# B&R Automation Studio project MotionTestBenchMaster (part 29)

```iecst
								VAR_RNS_SEQ.Device.PPB209_PID.PID_Enable := FALSE;                                      (* STEP: 0 PPB209*)
								VAR_RNS_SEQ.Device.PPB209_PID.PID_Mode := FALSE;
								VAR_RNS_SEQ.Device.PPB209_PID.Auto_SP_Value := 0;
								VAR_RNS_SEQ.Device.PPB209_PID.FIX_Value := 0;

								VAR_RNS_SEQ.Device.RVB202_PID.PID_Enable := FALSE;                                      (* STEP: 0 *)
								VAR_RNS_SEQ.Device.RVB202_PID.PID_Mode := FALSE;
								VAR_RNS_SEQ.Device.RVB202_PID.Auto_SP_Value := 0;
								VAR_RNS_SEQ.Device.RVB202_PID.FIX_Value := 0;

								VAR_RNS_SEQ.Device.FSB220.ALR := FALSE;                                                 (* STEP: 0 FSB220*)
								VAR_RNS_SEQ.Device.FSB220.WAIT_OFF := FALSE;
								VAR_RNS_SEQ.Device.FSB220.WAIT_ON := FALSE;

								VAR_RNS_SEQ.Device.LSB209.ALR := FALSE;                                                 (* STEP: 0 LSB209*)
								VAR_RNS_SEQ.Device.LSB209.WAIT_OFF := FALSE;
								VAR_RNS_SEQ.Device.LSB209.WAIT_ON := FALSE;

								VAR_RNS_SEQ.Device.LSB210.ALR := FALSE;                                                 (* STEP: 0 LSB210*)
								VAR_RNS_SEQ.Device.LSB210.WAIT_OFF := FALSE;
								VAR_RNS_SEQ.Device.LSB210.WAIT_ON := FALSE;

								VAR_RNS_SEQ.Device.LSB299.ALR := FALSE;                                                 (* STEP: 0 *)
								VAR_RNS_SEQ.Device.LSB299.WAIT_OFF := FALSE;
								VAR_RNS_SEQ.Device.LSB299.WAIT_ON := FALSE;

								VAR_RNS_SEQ.Device.FSB201.ALR := FALSE;                                                 (* STEP: 0 FSB201*)
								VAR_RNS_SEQ.Device.FSB201.WAIT_OFF := FALSE;
								VAR_RNS_SEQ.Device.FSB201.WAIT_ON := FALSE;

								VAR_RNS_SEQ.Device.FTB201.ALR_HighLimitEn := FALSE;                                     (* STEP: 0 FTB201*)
								VAR_RNS_SEQ.Device.FTB201.ALR_HighLimitSP := 0;
								VAR_RNS_SEQ.Device.FTB201.ALR_LowLimitEn := FALSE;
								VAR_RNS_SEQ.Device.FTB201.ALR_LowLimitSP := 0;
								VAR_RNS_SEQ.Device.FTB201.SP := 0;
								VAR_RNS_SEQ.Device.FTB201.CMP := 0;
								VAR_RNS_SEQ.Device.FTB201.MinDev := 0;
								VAR_RNS_SEQ.Device.FTB201.MaxDev := 0;

								VAR_RNS_SEQ.Device.FTB202.ALR_HighLimitEn := FALSE;                                     (* STEP: 0 FTB202*)
								VAR_RNS_SEQ.Device.FTB202.ALR_HighLimitSP := 0;
								VAR_RNS_SEQ.Device.FTB202.ALR_LowLimitEn := FALSE;
								VAR_RNS_SEQ.Device.FTB202.ALR_LowLimitSP := 0;
								VAR_RNS_SEQ.Device.FTB202.SP := 0;
								VAR_RNS_SEQ.Device.FTB202.CMP := 0;
								VAR_RNS_SEQ.Device.FTB202.MinDev := 0;
								VAR_RNS_SEQ.Device.FTB202.MaxDev := 0;

								VAR_RNS_SEQ.Device.PTB220.ALR_HighLimitEn := FALSE;                                     (* STEP: 0 PTB220*)
								VAR_RNS_SEQ.Device.PTB220.ALR_HighLimitSP := 0;
								VAR_RNS_SEQ.Device.PTB220.ALR_LowLimitEn := FALSE;
								VAR_RNS_SEQ.Device.PTB220.ALR_LowLimitSP := 0;
								VAR_RNS_SEQ.Device.PTB220.SP := 0;
								VAR_RNS_SEQ.Device.PTB220.CMP := 0;
								VAR_RNS_SEQ.Device.PTB220.MinDev := 0;
								VAR_RNS_SEQ.Device.PTB220.MaxDev := 0;

								VAR_RNS_SEQ.Device.PTB270.ALR_HighLimitEn := FALSE;                                     (* STEP: 0 PTB270*)
								VAR_RNS_SEQ.Device.PTB270.ALR_HighLimitSP := 0;
								VAR_RNS_SEQ.Device.PTB270.ALR_LowLimitEn := FALSE;
								VAR_RNS_SEQ.Device.PTB270.ALR_LowLimitSP := 0;
								VAR_RNS_SEQ.Device.PTB270.SP := 0;
								VAR_RNS_SEQ.Device.PTB270.CMP := 0;
								VAR_RNS_SEQ.Device.PTB270.MinDev := 0;
								VAR_RNS_SEQ.Device.PTB270.MaxDev := 0;

								VAR_RNS_SEQ.Device.LTB202.ALR_HighLimitEn := FALSE;                                     (* STEP: 0 LTB202*)
								VAR_RNS_SEQ.Device.LTB202.ALR_HighLimitSP := 0;
								VAR_RNS_SEQ.Device.LTB202.ALR_LowLimitEn := FALSE;
								VAR_RNS_SEQ.Device.LTB202.ALR_LowLimitSP := 0;
								VAR_RNS_SEQ.Device.LTB202.SP := 0;
								VAR_RNS_SEQ.Device.LTB202.CMP := 0;
								VAR_RNS_SEQ.Device.LTB202.MinDev := 0;
								VAR_RNS_SEQ.Device.LTB202.MaxDev := 0;

								VAR_RNS_SEQ.Device.PTB290.ALR_HighLimitEn := FALSE;                                     (* STEP: 0 PTB290*)
								VAR_RNS_SEQ.Device.PTB290.ALR_HighLimitSP := 0;
								VAR_RNS_SEQ.Device.PTB290.ALR_LowLimitEn := FALSE;
								VAR_RNS_SEQ.Device.PTB290.ALR_LowLimitSP := 0;
								VAR_RNS_SEQ.Device.PTB290.SP := 0;
								VAR_RNS_SEQ.Device.PTB290.CMP := 0;
								VAR_RNS_SEQ.Device.PTB290.MinDev := 0;
								VAR_RNS_SEQ.Device.PTB290.MaxDev := 0;

								VAR_RNS_SEQ.Mem.ContainersStop := TRUE;                                                (* STEP: 0 *)
								VAR_RNS_SEQ.Mem.ControlInsercion := FALSE;                                              (* STEP: 0 *)
								VAR_RNS_SEQ.Mem.ControlContinous := FALSE;                                              (* STEP: 0 *)
								VAR_RNS_SEQ.Mem.PBAbortEnable := FALSE;                                                 (* STEP: 0 PB Abort Sequence Enable*)
								VAR_RNS_SEQ.Mem.PBStopEnable := TRUE;                                                  (* STEP: 0 PB Stop Sequence Enable*)
								VAR_RNS_SEQ.Mem.PBStartEnable := FALSE;                                                  (* STEP: 0 PB Start Sequence Enable*)
								VAR_RNS_SEQ.Mem.ByPassed := FALSE;                                                      (* STEP: 0 *)
								VAR_RNS_SEQ.Mem.InsercionDevice := FALSE;                                               (* STEP: 0 *)
								VAR_RNS_SEQ.Mem.AirTreatmentControl := FALSE;                                           (* STEP: 0 *)
								VAR_RNS_SEQ.Mem.WaterTreatmentControl := FALSE;                                         (* STEP: 0 *)
								VAR_RNS_SEQ.Mem.SpeedReductionControl := FALSE;                                         (* STEP: 0 *)
								VAR_RNS_SEQ.Mem.ByPassRequest := FALSE;                                                 (* STEP: 0 *)
								VAR_RNS_SEQ.Mem.CopAfterCipRequest := FALSE;                                            (* STEP: 0 *)
								VAR_RNS_SEQ.Mem.NoBoNoSprayInsercion := FALSE;                                          (* STEP: 0 *)

								VAR_RNS_SEQ.ITC.WTT_ProductRequest := FALSE;                                            (* STEP: 0 *)
								VAR_RNS_SEQ.ITC.WTT_ProductionRunning := FALSE;

							36: (*MOTORIZATION - Waiting for Machine Stop - Disabling Axis*) //RnsDisable

								VAR_RNS_SEQ.Device.AVB224.AutoCnd := TRUE;                                              (* STEP: 0 AVB224*)
								VAR_RNS_SEQ.Device.AVB224.EnableCnd := FALSE;
								VAR_RNS_SEQ.Device.AVB228.AutoCnd := FALSE;                                             (* STEP: 0 AVB228*)
								VAR_RNS_SEQ.Device.AVB228.EnableCnd := FALSE;
								VAR_RNS_SEQ.Device.AVB234.AutoCnd := TRUE;                                              (* STEP: 0 AVB234*)
								VAR_RNS_SEQ.Device.AVB234.EnableCnd := FALSE;
								VAR_RNS_SEQ.Device.AVB261.AutoCnd := FALSE;                                             (* STEP: 0 AVB261*)
								VAR_RNS_SEQ.Device.AVB261.EnableCnd := FALSE;
								VAR_RNS_SEQ.Device.AVB264.AutoCnd := FALSE;                                             (* STEP: 0 AVB264*)
								VAR_RNS_SEQ.Device.AVB264.EnableCnd := FALSE;
								VAR_RNS_SEQ.Device.AVB265.AutoCnd := FALSE;                                             (* STEP: 0 AVB265*)
								VAR_RNS_SEQ.Device.AVB265.EnableCnd := FALSE;
								VAR_RNS_SEQ.Device.AVB266.AutoCnd := FALSE;                                             (* STEP: 0 AVB266*)
								VAR_RNS_SEQ.Device.AVB266.EnableCnd := FALSE;
								VAR_RNS_SEQ.Device.AVB267.AutoCnd := TRUE;                                              (* STEP: 0 AVB267*)
								VAR_RNS_SEQ.Device.AVB267.EnableCnd := FALSE;
								VAR_RNS_SEQ.Device.AVB268.AutoCnd := TRUE;                                              (* STEP: 0 AVB268*)
								VAR_RNS_SEQ.Device.AVB268.EnableCnd := FALSE;
								VAR_RNS_SEQ.Device.AVB273.AutoCnd := FALSE;                                             (* STEP: 0 AVB273*)
								VAR_RNS_SEQ.Device.AVB273.EnableCnd := FALSE;
								VAR_RNS_SEQ.Device.AVB294.AutoCnd := FALSE;                                             (* STEP: 0 AVB294*)
								VAR_RNS_SEQ.Device.AVB294.EnableCnd := FALSE;

								VAR_RNS_SEQ.Device.PPB209_PID.PID_Enable := FALSE;                                      (* STEP: 0 PPB209*)
								VAR_RNS_SEQ.Device.PPB209_PID.PID_Mode := FALSE;
								VAR_RNS_SEQ.Device.PPB209_PID.Auto_SP_Value := 0;
								VAR_RNS_SEQ.Device.PPB209_PID.FIX_Value := 0;

								VAR_RNS_SEQ.Device.RVB202_PID.PID_Enable := FALSE;                                      (* STEP: 0 *)
								VAR_RNS_SEQ.Device.RVB202_PID.PID_Mode := FALSE;
								VAR_RNS_SEQ.Device.RVB202_PID.Auto_SP_Value := 0;
								VAR_RNS_SEQ.Device.RVB202_PID.FIX_Value := 0;

								VAR_RNS_SEQ.Device.FSB220.ALR := FALSE;                                                 (* STEP: 0 FSB220*)
								VAR_RNS_SEQ.Device.FSB220.WAIT_OFF := FALSE;
								VAR_RNS_SEQ.Device.FSB220.WAIT_ON := FALSE;

								VAR_RNS_SEQ.Device.LSB209.ALR := FALSE;                                                 (* STEP: 0 LSB209*)
								VAR_RNS_SEQ.Device.LSB209.WAIT_OFF := FALSE;
								VAR_RNS_SEQ.Device.LSB209.WAIT_ON := FALSE;

								VAR_RNS_SEQ.Device.LSB210.ALR := FALSE;                                                 (* STEP: 0 LSB210*)
								VAR_RNS_SEQ.Device.LSB210.WAIT_OFF := FALSE;
								VAR_RNS_SEQ.Device.LSB210.WAIT_ON := FALSE;

								VAR_RNS_SEQ.Device.LSB299.ALR := FALSE;                                                 (* STEP: 0 *)
								VAR_RNS_SEQ.Device.LSB299.WAIT_OFF := FALSE;
								VAR_RNS_SEQ.Device.LSB299.WAIT_ON := FALSE;

								VAR_RNS_SEQ.Device.FSB201.ALR := FALSE;                                                 (* STEP: 0 FSB201*)
								VAR_RNS_SEQ.Device.FSB201.WAIT_OFF := FALSE;
								VAR_RNS_SEQ.Device.FSB201.WAIT_ON := FALSE;

								VAR_RNS_SEQ.Device.FTB201.ALR_HighLimitEn := FALSE;                                     (* STEP: 0 FTB201*)
								VAR_RNS_SEQ.Device.FTB201.ALR_HighLimitSP := 0;
								VAR_RNS_SEQ.Device.FTB201.ALR_LowLimitEn := FALSE;
								VAR_RNS_SEQ.Device.FTB201.ALR_LowLimitSP := 0;
								VAR_RNS_SEQ.Device.FTB201.SP := 0;
								VAR_RNS_SEQ.Device.FTB201.CMP := 0;
								VAR_RNS_SEQ.Device.FTB201.MinDev := 0;
								VAR_RNS_SEQ.Device.FTB201.MaxDev := 0;

								VAR_RNS_SEQ.Device.FTB202.ALR_HighLimitEn := FALSE;                                     (* STEP: 0 FTB202*)
								VAR_RNS_SEQ.Device.FTB202.ALR_HighLimitSP := 0;
								VAR_RNS_SEQ.Device.FTB202.ALR_LowLimitEn := FALSE;
								VAR_RNS_SEQ.Device.FTB202.ALR_LowLimitSP := 0;
								VAR_RNS_SEQ.Device.FTB202.SP := 0;
								VAR_RNS_SEQ.Device.FTB202.CMP := 0;
								VAR_RNS_SEQ.Device.FTB202.MinDev := 0;
								VAR_RNS_SEQ.Device.FTB202.MaxDev := 0;

								VAR_RNS_SEQ.Device.PTB220.ALR_HighLimitEn := FALSE;                                     (* STEP: 0 PTB220*)
								VAR_RNS_SEQ.Device.PTB220.ALR_HighLimitSP := 0;
								VAR_RNS_SEQ.Device.PTB220.ALR_LowLimitEn := FALSE;
								VAR_RNS_SEQ.Device.PTB220.ALR_LowLimitSP := 0;
								VAR_RNS_SEQ.Device.PTB220.SP := 0;
								VAR_RNS_SEQ.Device.PTB220.CMP := 0;
								VAR_RNS_SEQ.Device.PTB220.MinDev := 0;
								VAR_RNS_SEQ.Device.PTB220.MaxDev := 0;

								VAR_RNS_SEQ.Device.PTB270.ALR_HighLimitEn := FALSE;                                     (* STEP: 0 PTB270*)
								VAR_RNS_SEQ.Device.PTB270.ALR_HighLimitSP := 0;
								VAR_RNS_SEQ.Device.PTB270.ALR_LowLimitEn := FALSE;
								VAR_RNS_SEQ.Device.PTB270.ALR_LowLimitSP := 0;
								VAR_RNS_SEQ.Device.PTB270.SP := 0;
								VAR_RNS_SEQ.Device.PTB270.CMP := 0;
								VAR_RNS_SEQ.Device.PTB270.MinDev := 0;
								VAR_RNS_SEQ.Device.PTB270.MaxDev := 0;

								VAR_RNS_SEQ.Device.LTB202.ALR_HighLimitEn := FALSE;                                     (* STEP: 0 LTB202*)
								VAR_RNS_SEQ.Device.LTB202.ALR_HighLimitSP := 0;
								VAR_RNS_SEQ.Device.LTB202.ALR_LowLimitEn := FALSE;
								VAR_RNS_SEQ.Device.LTB202.ALR_LowLimitSP := 0;
								VAR_RNS_SEQ.Device.LTB202.SP := 0;
								VAR_RNS_SEQ.Device.LTB202.CMP := 0;
								VAR_RNS_SEQ.Device.LTB202.MinDev := 0;
								VAR_RNS_SEQ.Device.LTB202.MaxDev := 0;

								VAR_RNS_SEQ.Device.PTB290.ALR_HighLimitEn := FALSE;                                     (* STEP: 0 PTB290*)
								VAR_RNS_SEQ.Device.PTB290.ALR_HighLimitSP := 0;
								VAR_RNS_SEQ.Device.PTB290.ALR_LowLimitEn := FALSE;
								VAR_RNS_SEQ.Device.PTB290.ALR_LowLimitSP := 0;
								VAR_RNS_SEQ.Device.PTB290.SP := 0;
								VAR_RNS_SEQ.Device.PTB290.CMP := 0;
								VAR_RNS_SEQ.Device.PTB290.MinDev := 0;
								VAR_RNS_SEQ.Device.PTB290.MaxDev := 0;

								VAR_RNS_SEQ.Mem.ContainersStop := TRUE;                                                (* STEP: 0 *)
								VAR_RNS_SEQ.Mem.ControlInsercion := FALSE;                                              (* STEP: 0 *)
								VAR_RNS_SEQ.Mem.ControlContinous := FALSE;                                              (* STEP: 0 *)
								VAR_RNS_SEQ.Mem.PBAbortEnable := FALSE;                                                 (* STEP: 0 PB Abort Sequence Enable*)
								VAR_RNS_SEQ.Mem.PBStopEnable := TRUE;                                                  (* STEP: 0 PB Stop Sequence Enable*)
								VAR_RNS_SEQ.Mem.PBStartEnable := TRUE;                                                  (* STEP: 0 PB Start Sequence Enable*)
								VAR_RNS_SEQ.Mem.ByPassed := FALSE;                                                      (* STEP: 0 *)
								VAR_RNS_SEQ.Mem.InsercionDevice := FALSE;                                               (* STEP: 0 *)
								VAR_RNS_SEQ.Mem.AirTreatmentControl := FALSE;                                           (* STEP: 0 *)
								VAR_RNS_SEQ.Mem.WaterTreatmentControl := FALSE;                                         (* STEP: 0 *)
								VAR_RNS_SEQ.Mem.SpeedReductionControl := FALSE;                                         (* STEP: 0 *)
								VAR_RNS_SEQ.Mem.ByPassRequest := FALSE;                                                 (* STEP: 0 *)
								VAR_RNS_SEQ.Mem.CopAfterCipRequest := FALSE;                                            (* STEP: 0 *)
								VAR_RNS_SEQ.Mem.NoBoNoSprayInsercion := FALSE;                                          (* STEP: 0 *)

								VAR_RNS_SEQ.ITC.WTT_ProductRequest := FALSE;                                            (* STEP: 0 *)
								VAR_RNS_SEQ.ITC.WTT_ProductionRunning := FALSE;

						37..39: (* Spare Steps *)

						40: (* CIP - Wait Condition *)

                               VAR_RNS_SEQ.Device.AVB224.AutoCnd := FALSE;                                             (* STEP: 40 AVB224*)
                               VAR_RNS_SEQ.Device.AVB224.EnableCnd := FALSE;
                               VAR_RNS_SEQ.Device.AVB228.AutoCnd := FALSE;                                             (* STEP: 40 AVB228*)
                               VAR_RNS_SEQ.Device.AVB228.EnableCnd := FALSE;
                               VAR_RNS_SEQ.Device.AVB234.AutoCnd := FALSE;                                             (* STEP: 40 AVB234*)
                               VAR_RNS_SEQ.Device.AVB234.EnableCnd := FALSE;
                               VAR_RNS_SEQ.Device.AVB261.AutoCnd := TRUE;                                             (* STEP: 40 AVB261*)
                               VAR_RNS_SEQ.Device.AVB261.EnableCnd := FALSE;
                               VAR_RNS_SEQ.Device.AVB264.AutoCnd := FALSE;                                             (* STEP: 40 AVB264*)
                               VAR_RNS_SEQ.Device.AVB264.EnableCnd := FALSE;
                               VAR_RNS_SEQ.Device.AVB265.AutoCnd := FALSE;                                             (* STEP: 40 AVB265*)
                               VAR_RNS_SEQ.Device.AVB265.EnableCnd := FALSE;
                               VAR_RNS_SEQ.Device.AVB266.AutoCnd := TRUE;                                              (* STEP: 40 AVB266*)
                               VAR_RNS_SEQ.Device.AVB266.EnableCnd := FALSE;
                               VAR_RNS_SEQ.Device.AVB267.AutoCnd := FALSE;                                             (* STEP: 40 AVB267*)
                               VAR_RNS_SEQ.Device.AVB267.EnableCnd := FALSE;
                               VAR_RNS_SEQ.Device.AVB268.AutoCnd := FALSE;                                             (* STEP: 40 AVB268*)
                               VAR_RNS_SEQ.Device.AVB268.EnableCnd := FALSE;
                               VAR_RNS_SEQ.Device.AVB273.AutoCnd := FALSE;                                             (* STEP: 40 AVB273*)
                               VAR_RNS_SEQ.Device.AVB273.EnableCnd := FALSE;
                               VAR_RNS_SEQ.Device.AVB294.AutoCnd := FALSE;                                             (* STEP: 40 AVB294*)
                               VAR_RNS_SEQ.Device.AVB294.EnableCnd := FALSE;

                               VAR_RNS_SEQ.Device.PPB209_PID.PID_Enable := FALSE;                                      (* STEP: 40 PPB209*)
                               VAR_RNS_SEQ.Device.PPB209_PID.PID_Mode := FALSE;
                               VAR_RNS_SEQ.Device.PPB209_PID.Auto_SP_Value := 0;
                               VAR_RNS_SEQ.Device.PPB209_PID.FIX_Value := 0;

                               VAR_RNS_SEQ.Device.RVB202_PID.PID_Enable := TRUE;                                       (* STEP: 40 *)
                               VAR_RNS_SEQ.Device.RVB202_PID.PID_Mode := FALSE;
                               VAR_RNS_SEQ.Device.RVB202_PID.Auto_SP_Value := 0;
                               VAR_RNS_SEQ.Device.RVB202_PID.FIX_Value := HMI_PAM_1._093;

                               VAR_RNS_SEQ.Device.FSB220.ALR := FALSE;                                                 (* STEP: 40 FSB220*)
                               VAR_RNS_SEQ.Device.FSB220.WAIT_OFF := FALSE;
                               VAR_RNS_SEQ.Device.FSB220.WAIT_ON := FALSE;

                               VAR_RNS_SEQ.Device.LSB209.ALR := FALSE;                                                 (* STEP: 40 LSB209*)
                               VAR_RNS_SEQ.Device.LSB209.WAIT_OFF := FALSE;
                               VAR_RNS_SEQ.Device.LSB209.WAIT_ON := FALSE;

                               VAR_RNS_SEQ.Device.LSB210.ALR := FALSE;                                                 (* STEP: 40 LSB210*)
                               VAR_RNS_SEQ.Device.LSB210.WAIT_OFF := FALSE;
                               VAR_RNS_SEQ.Device.LSB210.WAIT_ON := FALSE;

                               VAR_RNS_SEQ.Device.LSB299.ALR := FALSE;                                                 (* STEP: 40 *)
                               VAR_RNS_SEQ.Device.LSB299.WAIT_OFF := FALSE;
                               VAR_RNS_SEQ.Device.LSB299.WAIT_ON := FALSE;

                               VAR_RNS_SEQ.Device.FSB201.ALR := FALSE;                                                 (* STEP: 40 FSB201*)
                               VAR_RNS_SEQ.Device.FSB201.WAIT_OFF := FALSE;
                               VAR_RNS_SEQ.Device.FSB201.WAIT_ON := FALSE;

                               VAR_RNS_SEQ.Device.FTB201.ALR_HighLimitEn := FALSE;                                     (* STEP: 40 FTB201*)
                               VAR_RNS_SEQ.Device.FTB201.ALR_HighLimitSP := 0;
                               VAR_RNS_SEQ.Device.FTB201.ALR_LowLimitEn := FALSE;
                               VAR_RNS_SEQ.Device.FTB201.ALR_LowLimitSP := 0;
                               VAR_RNS_SEQ.Device.FTB201.SP := 0;
                               VAR_RNS_SEQ.Device.FTB201.CMP := 0;
                               VAR_RNS_SEQ.Device.FTB201.MinDev := 0;
                               VAR_RNS_SEQ.Device.FTB201.MaxDev := 0;

                               VAR_RNS_SEQ.Device.FTB202.ALR_HighLimitEn := FALSE;                                     (* STEP: 40 FTB202*)
                               VAR_RNS_SEQ.Device.FTB202.ALR_HighLimitSP := 0;
                               VAR_RNS_SEQ.Device.FTB202.ALR_LowLimitEn := FALSE;
                               VAR_RNS_SEQ.Device.FTB202.ALR_LowLimitSP := 0;
                               VAR_RNS_SEQ.Device.FTB202.SP := 0;
                               VAR_RNS_SEQ.Device.FTB202.CMP := 0;
                               VAR_RNS_SEQ.Device.FTB202.MinDev := 0;
                               VAR_RNS_SEQ.Device.FTB202.MaxDev := 0;

                               VAR_RNS_SEQ.Device.PTB220.ALR_HighLimitEn := FALSE;                                     (* STEP: 40 PTB220*)
                               VAR_RNS_SEQ.Device.PTB220.ALR_HighLimitSP := 0;
                               VAR_RNS_SEQ.Device.PTB220.ALR_LowLimitEn := FALSE;
                               VAR_RNS_SEQ.Device.PTB220.ALR_LowLimitSP := 0;
                               VAR_RNS_SEQ.Device.PTB220.SP := 0;
                               VAR_RNS_SEQ.Device.PTB220.CMP := 0;
                               VAR_RNS_SEQ.Device.PTB220.MinDev := 0;
                               VAR_RNS_SEQ.Device.PTB220.MaxDev := 0;

                               VAR_RNS_SEQ.Device.PTB270.ALR_HighLimitEn := FALSE;                                     (* STEP: 40 PTB270*)
                               VAR_RNS_SEQ.Device.PTB270.ALR_HighLimitSP := 0;
                               VAR_RNS_SEQ.Device.PTB270.ALR_LowLimitEn := FALSE;
                               VAR_RNS_SEQ.Device.PTB270.ALR_LowLimitSP := 0;
                               VAR_RNS_SEQ.Device.PTB270.SP := 0;
                               VAR_RNS_SEQ.Device.PTB270.CMP := 0;
                               VAR_RNS_SEQ.Device.PTB270.MinDev := 0;
                               VAR_RNS_SEQ.Device.PTB270.MaxDev := 0;

                               VAR_RNS_SEQ.Device.LTB202.ALR_HighLimitEn := FALSE;                                     (* STEP: 40 LTB202*)
                               VAR_RNS_SEQ.Device.LTB202.ALR_HighLimitSP := 0;
                               VAR_RNS_SEQ.Device.LTB202.ALR_LowLimitEn := FALSE;
                               VAR_RNS_SEQ.Device.LTB202.ALR_LowLimitSP := 0;
                               VAR_RNS_SEQ.Device.LTB202.SP := 0;
                               VAR_RNS_SEQ.Device.LTB202.CMP := 0;
                               VAR_RNS_SEQ.Device.LTB202.MinDev := 0;
                               VAR_RNS_SEQ.Device.LTB202.MaxDev := 0;

                               VAR_RNS_SEQ.Device.PTB290.ALR_HighLimitEn := FALSE;                                     (* STEP: 40 PTB290*)
                               VAR_RNS_SEQ.Device.PTB290.ALR_HighLimitSP := 0;
                               VAR_RNS_SEQ.Device.PTB290.ALR_LowLimitEn := FALSE;
                               VAR_RNS_SEQ.Device.PTB290.ALR_LowLimitSP := 0;
                               VAR_RNS_SEQ.Device.PTB290.SP := 0;
                               VAR_RNS_SEQ.Device.PTB290.CMP := 0;
                               VAR_RNS_SEQ.Device.PTB290.MinDev := 0;
                               VAR_RNS_SEQ.Device.PTB290.MaxDev := 0;

                               VAR_RNS_SEQ.Mem.ContainersStop := TRUE;                                                 (* STEP: 40 *)
                               VAR_RNS_SEQ.Mem.ControlInsercion := FALSE;                                              (* STEP: 40 *)
                               VAR_RNS_SEQ.Mem.ControlContinous := FALSE;                                              (* STEP: 40 *)
                               VAR_RNS_SEQ.Mem.PBAbortEnable := FALSE;                                                 (* STEP: 40 PB Abort Sequence Enable*)
                               VAR_RNS_SEQ.Mem.PBStopEnable := TRUE;                                                   (* STEP: 40 PB Stop Sequence Enable*)
                               VAR_RNS_SEQ.Mem.PBStartEnable := FALSE;                                                 (* STEP: 40 PB Start Sequence Enable*)
                               VAR_RNS_SEQ.Mem.ByPassed := FALSE;                                                      (* STEP: 40 *)
                               VAR_RNS_SEQ.Mem.InsercionDevice := FALSE;                                               (* STEP: 40 *)
                               VAR_RNS_SEQ.Mem.AirTreatmentControl := FALSE;                                           (* STEP: 40 *)
                               VAR_RNS_SEQ.Mem.WaterTreatmentControl := FALSE;                                         (* STEP: 40 *)
                               VAR_RNS_SEQ.Mem.SpeedReductionControl := FALSE;                                         (* STEP: 40 *)
                               VAR_RNS_SEQ.Mem.ByPassRequest := FALSE;                                                 (* STEP: 40 *)
                               VAR_RNS_SEQ.Mem.CopAfterCipRequest := FALSE;                                            (* STEP: 40 *)
                               VAR_RNS_SEQ.Mem.NoBoNoSprayInsercion := FALSE;                                          (* STEP: 40 *)

                               VAR_RNS_SEQ.ITC.WTT_ProductRequest := TRUE;                                             (* STEP: 40 *)
                               VAR_RNS_SEQ.ITC.WTT_ProductionRunning := FALSE;                                         (* STEP: 40 *)

                       41: (* CIP - Execution *)

                               VAR_RNS_SEQ.Device.AVB224.AutoCnd := FALSE;                                             (* STEP: 41 AVB224*)
                               VAR_RNS_SEQ.Device.AVB224.EnableCnd := FALSE;
                               VAR_RNS_SEQ.Device.AVB228.AutoCnd := FALSE;                                             (* STEP: 41 AVB228*)
                               VAR_RNS_SEQ.Device.AVB228.EnableCnd := FALSE;
                               VAR_RNS_SEQ.Device.AVB234.AutoCnd := FALSE;                                             (* STEP: 41 AVB234*)
                               VAR_RNS_SEQ.Device.AVB234.EnableCnd := FALSE;
                               VAR_RNS_SEQ.Device.AVB261.AutoCnd := TRUE;                                              (* STEP: 41 AVB261*)
                               VAR_RNS_SEQ.Device.AVB261.EnableCnd := FALSE;
                               VAR_RNS_SEQ.Device.AVB264.AutoCnd := FALSE;                                             (* STEP: 41 AVB264*)
                               VAR_RNS_SEQ.Device.AVB264.EnableCnd := FALSE;
                               VAR_RNS_SEQ.Device.AVB265.AutoCnd := TRUE;                                              (* STEP: 41 AVB265*)
                               VAR_RNS_SEQ.Device.AVB265.EnableCnd := FALSE;
                               VAR_RNS_SEQ.Device.AVB266.AutoCnd := TRUE;                                              (* STEP: 41 AVB266*)
                               VAR_RNS_SEQ.Device.AVB266.EnableCnd := FALSE;
                               VAR_RNS_SEQ.Device.AVB267.AutoCnd := TRUE;                                              (* STEP: 41 AVB267*)
                               VAR_RNS_SEQ.Device.AVB267.EnableCnd := FALSE;
                               VAR_RNS_SEQ.Device.AVB268.AutoCnd := TRUE;                                              (* STEP: 41 AVB268*)
                               VAR_RNS_SEQ.Device.AVB268.EnableCnd := TRUE;
                               VAR_RNS_SEQ.Device.AVB273.AutoCnd := FALSE;                                             (* STEP: 41 AVB273*)
                               VAR_RNS_SEQ.Device.AVB273.EnableCnd := FALSE;
                               VAR_RNS_SEQ.Device.AVB294.AutoCnd := TRUE;                                              (* STEP: 41 AVB294*)
                               VAR_RNS_SEQ.Device.AVB294.EnableCnd := TRUE;

                               VAR_RNS_SEQ.Device.PPB209_PID.PID_Enable := FALSE;                                      (* STEP: 41 PPB209*)
                               VAR_RNS_SEQ.Device.PPB209_PID.PID_Mode := FALSE;
                               VAR_RNS_SEQ.Device.PPB209_PID.Auto_SP_Value := 0;
                               VAR_RNS_SEQ.Device.PPB209_PID.FIX_Value := 0;

                               VAR_RNS_SEQ.Device.RVB202_PID.PID_Enable := TRUE;                                       (* STEP: 41 *)
                               VAR_RNS_SEQ.Device.RVB202_PID.PID_Mode := FALSE;
                               VAR_RNS_SEQ.Device.RVB202_PID.Auto_SP_Value := 0;
                               VAR_RNS_SEQ.Device.RVB202_PID.FIX_Value := HMI_PAM_1._093;

                               VAR_RNS_SEQ.Device.FSB220.ALR := FALSE;                                                 (* STEP: 41 FSB220*)
                               VAR_RNS_SEQ.Device.FSB220.WAIT_OFF := FALSE;
                               VAR_RNS_SEQ.Device.FSB220.WAIT_ON := FALSE;

                               VAR_RNS_SEQ.Device.LSB209.ALR := FALSE;                                                 (* STEP: 41 LSB209*)
                               VAR_RNS_SEQ.Device.LSB209.WAIT_OFF := FALSE;
                               VAR_RNS_SEQ.Device.LSB209.WAIT_ON := FALSE;

                               VAR_RNS_SEQ.Device.LSB210.ALR := FALSE;                                                 (* STEP: 41 LSB210*)
                               VAR_RNS_SEQ.Device.LSB210.WAIT_OFF := FALSE;
                               VAR_RNS_SEQ.Device.LSB210.WAIT_ON := FALSE;

                               VAR_RNS_SEQ.Device.LSB299.ALR := FALSE;                                                 (* STEP: 41 *)
                               VAR_RNS_SEQ.Device.LSB299.WAIT_OFF := FALSE;
                               VAR_RNS_SEQ.Device.LSB299.WAIT_ON := FALSE;

                               VAR_RNS_SEQ.Device.FSB201.ALR := FALSE;                                                 (* STEP: 41 FSB201*)
                               VAR_RNS_SEQ.Device.FSB201.WAIT_OFF := FALSE;
                               VAR_RNS_SEQ.Device.FSB201.WAIT_ON := FALSE;

                               VAR_RNS_SEQ.Device.FTB201.ALR_HighLimitEn := FALSE;                                     (* STEP: 41 FTB201*)
                               VAR_RNS_SEQ.Device.FTB201.ALR_HighLimitSP := 0;
                               VAR_RNS_SEQ.Device.FTB201.ALR_LowLimitEn := FALSE;
                               VAR_RNS_SEQ.Device.FTB201.ALR_LowLimitSP := 0;
                               VAR_RNS_SEQ.Device.FTB201.SP := 0;
                               VAR_RNS_SEQ.Device.FTB201.CMP := 0;
                               VAR_RNS_SEQ.Device.FTB201.MinDev := 0;
                               VAR_RNS_SEQ.Device.FTB201.MaxDev := 0;

                               VAR_RNS_SEQ.Device.FTB202.ALR_HighLimitEn := FALSE;                                     (* STEP: 41 FTB202*)
                               VAR_RNS_SEQ.Device.FTB202.ALR_HighLimitSP := 0;
                               VAR_RNS_SEQ.Device.FTB202.ALR_LowLimitEn := FALSE;
                               VAR_RNS_SEQ.Device.FTB202.ALR_LowLimitSP := 0;
                               VAR_RNS_SEQ.Device.FTB202.SP := 0;
                               VAR_RNS_SEQ.Device.FTB202.CMP := 0;
                               VAR_RNS_SEQ.Device.FTB202.MinDev := 0;
                               VAR_RNS_SEQ.Device.FTB202.MaxDev := 0;

                               VAR_RNS_SEQ.Device.PTB220.ALR_HighLimitEn := FALSE;                                     (* STEP: 41 PTB220*)
                               VAR_RNS_SEQ.Device.PTB220.ALR_HighLimitSP := 0;
                               VAR_RNS_SEQ.Device.PTB220.ALR_LowLimitEn := FALSE;
                               VAR_RNS_SEQ.Device.PTB220.ALR_LowLimitSP := 0;
                               VAR_RNS_SEQ.Device.PTB220.SP := 0;
                               VAR_RNS_SEQ.Device.PTB220.CMP := 0;
                               VAR_RNS_SEQ.Device.PTB220.MinDev := 0;
                               VAR_RNS_SEQ.Device.PTB220.MaxDev := 0;

                               VAR_RNS_SEQ.Device.PTB270.ALR_HighLimitEn := FALSE;                                     (* STEP: 41 PTB270*)
                               VAR_RNS_SEQ.Device.PTB270.ALR_HighLimitSP := 0;
                               VAR_RNS_SEQ.Device.PTB270.ALR_LowLimitEn := FALSE;
                               VAR_RNS_SEQ.Device.PTB270.ALR_LowLimitSP := 0;
                               VAR_RNS_SEQ.Device.PTB270.SP := 0;
                               VAR_RNS_SEQ.Device.PTB270.CMP := 0;
                               VAR_RNS_SEQ.Device.PTB270.MinDev := 0;
                               VAR_RNS_SEQ.Device.PTB270.MaxDev := 0;

                               VAR_RNS_SEQ.Device.LTB202.ALR_HighLimitEn := TRUE;                                      (* STEP: 41 LTB202*)
                               VAR_RNS_SEQ.Device.LTB202.ALR_HighLimitSP := 80;
                               VAR_RNS_SEQ.Device.LTB202.ALR_LowLimitEn := FALSE;
                               VAR_RNS_SEQ.Device.LTB202.ALR_LowLimitSP := 0;
                               VAR_RNS_SEQ.Device.LTB202.SP := 0;
                               VAR_RNS_SEQ.Device.LTB202.CMP := 0;
                               VAR_RNS_SEQ.Device.LTB202.MinDev := 0;
                               VAR_RNS_SEQ.Device.LTB202.MaxDev := 0;

                               VAR_RNS_SEQ.Device.PTB290.ALR_HighLimitEn := FALSE;                                     (* STEP: 41 PTB290*)
                               VAR_RNS_SEQ.Device.PTB290.ALR_HighLimitSP := 0;
                               VAR_RNS_SEQ.Device.PTB290.ALR_LowLimitEn := FALSE;
                               VAR_RNS_SEQ.Device.PTB290.ALR_LowLimitSP := 0;
                               VAR_RNS_SEQ.Device.PTB290.SP := 0;
                               VAR_RNS_SEQ.Device.PTB290.CMP := 0;
                               VAR_RNS_SEQ.Device.PTB290.MinDev := 0;
                               VAR_RNS_SEQ.Device.PTB290.MaxDev := 0;

                               VAR_RNS_SEQ.Mem.ContainersStop := TRUE;                                                 (* STEP: 41 *)
                               VAR_RNS_SEQ.Mem.ControlInsercion := FALSE;                                              (* STEP: 41 *)
                               VAR_RNS_SEQ.Mem.ControlContinous := FALSE;                                              (* STEP: 41 *)
                               VAR_RNS_SEQ.Mem.PBAbortEnable := FALSE;                                                 (* STEP: 41 PB Abort Sequence Enable*)
                               VAR_RNS_SEQ.Mem.PBStopEnable := TRUE;                                                   (* STEP: 41 PB Stop Sequence Enable*)
                               VAR_RNS_SEQ.Mem.PBStartEnable := FALSE;                                                 (* STEP: 41 PB Start Sequence Enable*)
                               VAR_RNS_SEQ.Mem.ByPassed := FALSE;                                                      (* STEP: 41 *)
                               VAR_RNS_SEQ.Mem.InsercionDevice := FALSE;                                               (* STEP: 41 *)
                               VAR_RNS_SEQ.Mem.AirTreatmentControl := FALSE;                                           (* STEP: 41 *)
                               VAR_RNS_SEQ.Mem.WaterTreatmentControl := FALSE;                                         (* STEP: 41 *)
                               VAR_RNS_SEQ.Mem.SpeedReductionControl := TRUE;                                         (* STEP: 41 *)
                               VAR_RNS_SEQ.Mem.ByPassRequest := FALSE;                                                 (* STEP: 41 *)
                               VAR_RNS_SEQ.Mem.CopAfterCipRequest := FALSE;                                            (* STEP: 41 *)
                               VAR_RNS_SEQ.Mem.NoBoNoSprayInsercion := FALSE;                                          (* STEP: 41 *)

                               VAR_RNS_SEQ.ITC.WTT_ProductRequest := TRUE;                                             (* STEP: 41 *)
                               VAR_RNS_SEQ.ITC.WTT_ProductionRunning := FALSE;                                         (* STEP: 41 *)

                       42..45: (* Spare Steps *)

		46: (*MOTORIZATION - Waiting for Machine Stop - Disabling Axis*) //RnsDisable

			VAR_RNS_SEQ.Device.AVB224.AutoCnd := TRUE;                                              (* STEP: 0 AVB224*)
			VAR_RNS_SEQ.Device.AVB224.EnableCnd := FALSE;
			VAR_RNS_SEQ.Device.AVB228.AutoCnd := FALSE;                                             (* STEP: 0 AVB228*)
			VAR_RNS_SEQ.Device.AVB228.EnableCnd := FALSE;
			VAR_RNS_SEQ.Device.AVB234.AutoCnd := TRUE;                                              (* STEP: 0 AVB234*)
			VAR_RNS_SEQ.Device.AVB234.EnableCnd := FALSE;
			VAR_RNS_SEQ.Device.AVB261.AutoCnd := FALSE;                                             (* STEP: 0 AVB261*)
			VAR_RNS_SEQ.Device.AVB261.EnableCnd := FALSE;
			VAR_RNS_SEQ.Device.AVB264.AutoCnd := FALSE;                                             (* STEP: 0 AVB264*)
			VAR_RNS_SEQ.Device.AVB264.EnableCnd := FALSE;
			VAR_RNS_SEQ.Device.AVB265.AutoCnd := FALSE;                                             (* STEP: 0 AVB265*)
			VAR_RNS_SEQ.Device.AVB265.EnableCnd := FALSE;
			VAR_RNS_SEQ.Device.AVB266.AutoCnd := FALSE;                                             (* STEP: 0 AVB266*)
			VAR_RNS_SEQ.Device.AVB266.EnableCnd := FALSE;
			VAR_RNS_SEQ.Device.AVB267.AutoCnd := TRUE;                                              (* STEP: 0 AVB267*)
			VAR_RNS_SEQ.Device.AVB267.EnableCnd := FALSE;
			VAR_RNS_SEQ.Device.AVB268.AutoCnd := TRUE;                                              (* STEP: 0 AVB268*)
			VAR_RNS_SEQ.Device.AVB268.EnableCnd := FALSE;
			VAR_RNS_SEQ.Device.AVB273.AutoCnd := FALSE;                                             (* STEP: 0 AVB273*)
			VAR_RNS_SEQ.Device.AVB273.EnableCnd := FALSE;
			VAR_RNS_SEQ.Device.AVB294.AutoCnd := FALSE;                                             (* STEP: 0 AVB294*)
			VAR_RNS_SEQ.Device.AVB294.EnableCnd := FALSE;

			VAR_RNS_SEQ.Device.PPB209_PID.PID_Enable := FALSE;                                      (* STEP: 0 PPB209*)
			VAR_RNS_SEQ.Device.PPB209_PID.PID_Mode := FALSE;
			VAR_RNS_SEQ.Device.PPB209_PID.Auto_SP_Value := 0;
			VAR_RNS_SEQ.Device.PPB209_PID.FIX_Value := 0;

			VAR_RNS_SEQ.Device.RVB202_PID.PID_Enable := FALSE;                                      (* STEP: 0 *)
			VAR_RNS_SEQ.Device.RVB202_PID.PID_Mode := FALSE;
			VAR_RNS_SEQ.Device.RVB202_PID.Auto_SP_Value := 0;
			VAR_RNS_SEQ.Device.RVB202_PID.FIX_Value := 0;

			VAR_RNS_SEQ.Device.FSB220.ALR := FALSE;                                                 (* STEP: 0 FSB220*)
			VAR_RNS_SEQ.Device.FSB220.WAIT_OFF := FALSE;
			VAR_RNS_SEQ.Device.FSB220.WAIT_ON := FALSE;

			VAR_RNS_SEQ.Device.LSB209.ALR := FALSE;                                                 (* STEP: 0 LSB209*)
			VAR_RNS_SEQ.Device.LSB209.WAIT_OFF := FALSE;
			VAR_RNS_SEQ.Device.LSB209.WAIT_ON := FALSE;

			VAR_RNS_SEQ.Device.LSB210.ALR := FALSE;                                                 (* STEP: 0 LSB210*)
			VAR_RNS_SEQ.Device.LSB210.WAIT_OFF := FALSE;
			VAR_RNS_SEQ.Device.LSB210.WAIT_ON := FALSE;

			VAR_RNS_SEQ.Device.LSB299.ALR := FALSE;                                                 (* STEP: 0 *)
			VAR_RNS_SEQ.Device.LSB299.WAIT_OFF := FALSE;
			VAR_RNS_SEQ.Device.LSB299.WAIT_ON := FALSE;

			VAR_RNS_SEQ.Device.FSB201.ALR := FALSE;                                                 (* STEP: 0 FSB201*)
			VAR_RNS_SEQ.Device.FSB201.WAIT_OFF := FALSE;
			VAR_RNS_SEQ.Device.FSB201.WAIT_ON := FALSE;

			VAR_RNS_SEQ.Device.FTB201.ALR_HighLimitEn := FALSE;                                     (* STEP: 0 FTB201*)
			VAR_RNS_SEQ.Device.FTB201.ALR_HighLimitSP := 0;
			VAR_RNS_SEQ.Device.FTB201.ALR_LowLimitEn := FALSE;
			VAR_RNS_SEQ.Device.FTB201.ALR_LowLimitSP := 0;
			VAR_RNS_SEQ.Device.FTB201.SP := 0;
			VAR_RNS_SEQ.Device.FTB201.CMP := 0;
			VAR_RNS_SEQ.Device.FTB201.MinDev := 0;
			VAR_RNS_SEQ.Device.FTB201.MaxDev := 0;

			VAR_RNS_SEQ.Device.FTB202.ALR_HighLimitEn := FALSE;                                     (* STEP: 0 FTB202*)
			VAR_RNS_SEQ.Device.FTB202.ALR_HighLimitSP := 0;
			VAR_RNS_SEQ.Device.FTB202.ALR_LowLimitEn := FALSE;
			VAR_RNS_SEQ.Device.FTB202.ALR_LowLimitSP := 0;
			VAR_RNS_SEQ.Device.FTB202.SP := 0;
			VAR_RNS_SEQ.Device.FTB202.CMP := 0;
			VAR_RNS_SEQ.Device.FTB202.MinDev := 0;
			VAR_RNS_SEQ.Device.FTB202.MaxDev := 0;

			VAR_RNS_SEQ.Device.PTB220.ALR_HighLimitEn := FALSE;                                     (* STEP: 0 PTB220*)
			VAR_RNS_SEQ.Device.PTB220.ALR_HighLimitSP := 0;
			VAR_RNS_SEQ.Device.PTB220.ALR_LowLimitEn := FALSE;
			VAR_RNS_SEQ.Device.PTB220.ALR_LowLimitSP := 0;
			VAR_RNS_SEQ.Device.PTB220.SP := 0;
			VAR_RNS_SEQ.Device.PTB220.CMP := 0;
			VAR_RNS_SEQ.Device.PTB220.MinDev := 0;
			VAR_RNS_SEQ.Device.PTB220.MaxDev := 0;

			VAR_RNS_SEQ.Device.PTB270.ALR_HighLimitEn := FALSE;                                     (* STEP: 0 PTB270*)
			VAR_RNS_SEQ.Device.PTB270.ALR_HighLimitSP := 0;
			VAR_RNS_SEQ.Device.PTB270.ALR_LowLimitEn := FALSE;
			VAR_RNS_SEQ.Device.PTB270.ALR_LowLimitSP := 0;
			VAR_RNS_SEQ.Device.PTB270.SP := 0;
			VAR_RNS_SEQ.Device.PTB270.CMP := 0;
			VAR_RNS_SEQ.Device.PTB270.MinDev := 0;
			VAR_RNS_SEQ.Device.PTB270.MaxDev := 0;

			VAR_RNS_SEQ.Device.LTB202.ALR_HighLimitEn := FALSE;                                     (* STEP: 0 LTB202*)
			VAR_RNS_SEQ.Device.LTB202.ALR_HighLimitSP := 0;
			VAR_RNS_SEQ.Device.LTB202.ALR_LowLimitEn := FALSE;
			VAR_RNS_SEQ.Device.LTB202.ALR_LowLimitSP := 0;
			VAR_RNS_SEQ.Device.LTB202.SP := 0;
			VAR_RNS_SEQ.Device.LTB202.CMP := 0;
			VAR_RNS_SEQ.Device.LTB202.MinDev := 0;
			VAR_RNS_SEQ.Device.LTB202.MaxDev := 0;

			VAR_RNS_SEQ.Device.PTB290.ALR_HighLimitEn := FALSE;                                     (* STEP: 0 PTB290*)
			VAR_RNS_SEQ.Device.PTB290.ALR_HighLimitSP := 0;
			VAR_RNS_SEQ.Device.PTB290.ALR_LowLimitEn := FALSE;
			VAR_RNS_SEQ.Device.PTB290.ALR_LowLimitSP := 0;
			VAR_RNS_SEQ.Device.PTB290.SP := 0;
			VAR_RNS_SEQ.Device.PTB290.CMP := 0;
			VAR_RNS_SEQ.Device.PTB290.MinDev := 0;
			VAR_RNS_SEQ.Device.PTB290.MaxDev := 0;

			VAR_RNS_SEQ.Mem.ContainersStop := TRUE;                                                (* STEP: 0 *)
			VAR_RNS_SEQ.Mem.ControlInsercion := FALSE;                                              (* STEP: 0 *)
			VAR_RNS_SEQ.Mem.ControlContinous := FALSE;                                              (* STEP: 0 *)
			VAR_RNS_SEQ.Mem.PBAbortEnable := FALSE;                                                 (* STEP: 0 PB Abort Sequence Enable*)
			VAR_RNS_SEQ.Mem.PBStopEnable := TRUE;                                                  (* STEP: 0 PB Stop Sequence Enable*)
			VAR_RNS_SEQ.Mem.PBStartEnable := TRUE;                                                  (* STEP: 0 PB Start Sequence Enable*)
			VAR_RNS_SEQ.Mem.ByPassed := FALSE;                                                      (* STEP: 0 *)
			VAR_RNS_SEQ.Mem.InsercionDevice := FALSE;                                               (* STEP: 0 *)
			VAR_RNS_SEQ.Mem.AirTreatmentControl := FALSE;                                           (* STEP: 0 *)
			VAR_RNS_SEQ.Mem.WaterTreatmentControl := FALSE;                                         (* STEP: 0 *)
			VAR_RNS_SEQ.Mem.SpeedReductionControl := FALSE;                                         (* STEP: 0 *)
			VAR_RNS_SEQ.Mem.ByPassRequest := FALSE;                                                 (* STEP: 0 *)
			VAR_RNS_SEQ.Mem.CopAfterCipRequest := FALSE;                                            (* STEP: 0 *)
			VAR_RNS_SEQ.Mem.NoBoNoSprayInsercion := FALSE;                                          (* STEP: 0 *)

			VAR_RNS_SEQ.ITC.WTT_ProductRequest := FALSE;                                            (* STEP: 0 *)
			VAR_RNS_SEQ.ITC.WTT_ProductionRunning := FALSE;

		47: (* CIP - Drain *)

                               VAR_RNS_SEQ.Device.AVB224.AutoCnd := TRUE;                                              (* STEP: 47 AVB224*)
                               VAR_RNS_SEQ.Device.AVB224.EnableCnd := FALSE;
                               VAR_RNS_SEQ.Device.AVB228.AutoCnd := FALSE;                                             (* STEP: 47 AVB228*)
                               VAR_RNS_SEQ.Device.AVB228.EnableCnd := FALSE;
                               VAR_RNS_SEQ.Device.AVB234.AutoCnd := FALSE;                                             (* STEP: 47 AVB234*)
                               VAR_RNS_SEQ.Device.AVB234.EnableCnd := FALSE;
                               VAR_RNS_SEQ.Device.AVB261.AutoCnd := FALSE;                                             (* STEP: 47 AVB261*)
                               VAR_RNS_SEQ.Device.AVB261.EnableCnd := FALSE;
                               VAR_RNS_SEQ.Device.AVB264.AutoCnd := FALSE;                                             (* STEP: 47 AVB264*)
                               VAR_RNS_SEQ.Device.AVB264.EnableCnd := FALSE;
                               VAR_RNS_SEQ.Device.AVB265.AutoCnd := TRUE;                                              (* STEP: 47 AVB265*)
                               VAR_RNS_SEQ.Device.AVB265.EnableCnd := FALSE;
                               VAR_RNS_SEQ.Device.AVB266.AutoCnd := TRUE;                                              (* STEP: 47 AVB266*)
                               VAR_RNS_SEQ.Device.AVB266.EnableCnd := FALSE;
                               VAR_RNS_SEQ.Device.AVB267.AutoCnd := TRUE;                                              (* STEP: 47 AVB267*)
                               VAR_RNS_SEQ.Device.AVB267.EnableCnd := FALSE;
                               VAR_RNS_SEQ.Device.AVB268.AutoCnd := TRUE;                                              (* STEP: 47 AVB268*)
                               VAR_RNS_SEQ.Device.AVB268.EnableCnd := FALSE;
                               VAR_RNS_SEQ.Device.AVB273.AutoCnd := FALSE;                                             (* STEP: 47 AVB273*)
                               VAR_RNS_SEQ.Device.AVB273.EnableCnd := FALSE;
                               VAR_RNS_SEQ.Device.AVB294.AutoCnd := FALSE;                                             (* STEP: 47 AVB294*)
                               VAR_RNS_SEQ.Device.AVB294.EnableCnd := FALSE;

                               VAR_RNS_SEQ.Device.PPB209_PID.PID_Enable := FALSE;                                      (* STEP: 47 PPB209*)
                               VAR_RNS_SEQ.Device.PPB209_PID.PID_Mode := FALSE;
                               VAR_RNS_SEQ.Device.PPB209_PID.Auto_SP_Value := 0;
                               VAR_RNS_SEQ.Device.PPB209_PID.FIX_Value := 0;

                               VAR_RNS_SEQ.Device.RVB202_PID.PID_Enable := FALSE;                                      (* STEP: 47 *)
                               VAR_RNS_SEQ.Device.RVB202_PID.PID_Mode := FALSE;
                               VAR_RNS_SEQ.Device.RVB202_PID.Auto_SP_Value := 0;
                               VAR_RNS_SEQ.Device.RVB202_PID.FIX_Value := 0;

                               VAR_RNS_SEQ.Device.FSB220.ALR := FALSE;                                                 (* STEP: 47 FSB220*)
                               VAR_RNS_SEQ.Device.FSB220.WAIT_OFF := FALSE;
                               VAR_RNS_SEQ.Device.FSB220.WAIT_ON := FALSE;

                               VAR_RNS_SEQ.Device.LSB209.ALR := FALSE;                                                 (* STEP: 47 LSB209*)
                               VAR_RNS_SEQ.Device.LSB209.WAIT_OFF := FALSE;
                               VAR_RNS_SEQ.Device.LSB209.WAIT_ON := FALSE;

                               VAR_RNS_SEQ.Device.LSB210.ALR := FALSE;                                                 (* STEP: 47 LSB210*)
                               VAR_RNS_SEQ.Device.LSB210.WAIT_OFF := FALSE;
                               VAR_RNS_SEQ.Device.LSB210.WAIT_ON := FALSE;

                               VAR_RNS_SEQ.Device.LSB299.ALR := FALSE;                                                 (* STEP: 47 *)
                               VAR_RNS_SEQ.Device.LSB299.WAIT_OFF := FALSE;
                               VAR_RNS_SEQ.Device.LSB299.WAIT_ON := FALSE;

                               VAR_RNS_SEQ.Device.FSB201.ALR := FALSE;                                                 (* STEP: 47 FSB201*)
                               VAR_RNS_SEQ.Device.FSB201.WAIT_OFF := FALSE;
                               VAR_RNS_SEQ.Device.FSB201.WAIT_ON := FALSE;

                               VAR_RNS_SEQ.Device.FTB201.ALR_HighLimitEn := FALSE;                                     (* STEP: 47 FTB201*)
                               VAR_RNS_SEQ.Device.FTB201.ALR_HighLimitSP := 0;
                               VAR_RNS_SEQ.Device.FTB201.ALR_LowLimitEn := FALSE;
                               VAR_RNS_SEQ.Device.FTB201.ALR_LowLimitSP := 0;
                               VAR_RNS_SEQ.Device.FTB201.SP := 0;
                               VAR_RNS_SEQ.Device.FTB201.CMP := 0;
                               VAR_RNS_SEQ.Device.FTB201.MinDev := 0;
                               VAR_RNS_SEQ.Device.FTB201.MaxDev := 0;

                               VAR_RNS_SEQ.Device.FTB202.ALR_HighLimitEn := FALSE;                                     (* STEP: 47 FTB202*)
                               VAR_RNS_SEQ.Device.FTB202.ALR_HighLimitSP := 0;
                               VAR_RNS_SEQ.Device.FTB202.ALR_LowLimitEn := FALSE;
                               VAR_RNS_SEQ.Device.FTB202.ALR_LowLimitSP := 0;
                               VAR_RNS_SEQ.Device.FTB202.SP := 0;
                               VAR_RNS_SEQ.Device.FTB202.CMP := 0;
                               VAR_RNS_SEQ.Device.FTB202.MinDev := 0;
                               VAR_RNS_SEQ.Device.FTB202.MaxDev := 0;

                               VAR_RNS_SEQ.Device.PTB220.ALR_HighLimitEn := FALSE;                                     (* STEP: 47 PTB220*)
                               VAR_RNS_SEQ.Device.PTB220.ALR_HighLimitSP := 0;
                               VAR_RNS_SEQ.Device.PTB220.ALR_LowLimitEn := FALSE;
                               VAR_RNS_SEQ.Device.PTB220.ALR_LowLimitSP := 0;
                               VAR_RNS_SEQ.Device.PTB220.SP := 0;
                               VAR_RNS_SEQ.Device.PTB220.CMP := 0;
                               VAR_RNS_SEQ.Device.PTB220.MinDev := 0;
                               VAR_RNS_SEQ.Device.PTB220.MaxDev := 0;

                               VAR_RNS_SEQ.Device.PTB270.ALR_HighLimitEn := FALSE;                                     (* STEP: 47 PTB270*)
                               VAR_RNS_SEQ.Device.PTB270.ALR_HighLimitSP := 0;
                               VAR_RNS_SEQ.Device.PTB270.ALR_LowLimitEn := FALSE;
                               VAR_RNS_SEQ.Device.PTB270.ALR_LowLimitSP := 0;
                               VAR_RNS_SEQ.Device.PTB270.SP := 0;
                               VAR_RNS_SEQ.Device.PTB270.CMP := 0;
                               VAR_RNS_SEQ.Device.PTB270.MinDev := 0;
                               VAR_RNS_SEQ.Device.PTB270.MaxDev := 0;

                               VAR_RNS_SEQ.Device.LTB202.ALR_HighLimitEn := FALSE;                                     (* STEP: 47 LTB202*)
                               VAR_RNS_SEQ.Device.LTB202.ALR_HighLimitSP := 0;
                               VAR_RNS_SEQ.Device.LTB202.ALR_LowLimitEn := FALSE;
                               VAR_RNS_SEQ.Device.LTB202.ALR_LowLimitSP := 0;
                               VAR_RNS_SEQ.Device.LTB202.SP := 0;
                               VAR_RNS_SEQ.Device.LTB202.CMP := 0;
                               VAR_RNS_SEQ.Device.LTB202.MinDev := 0;
                               VAR_RNS_SEQ.Device.LTB202.MaxDev := 0;

                               VAR_RNS_SEQ.Device.PTB290.ALR_HighLimitEn := FALSE;                                     (* STEP: 47 PTB290*)
                               VAR_RNS_SEQ.Device.PTB290.ALR_HighLimitSP := 0;
                               VAR_RNS_SEQ.Device.PTB290.ALR_LowLimitEn := FALSE;
                               VAR_RNS_SEQ.Device.PTB290.ALR_LowLimitSP := 0;
                               VAR_RNS_SEQ.Device.PTB290.SP := 0;
                               VAR_RNS_SEQ.Device.PTB290.CMP := 0;
                               VAR_RNS_SEQ.Device.PTB290.MinDev := 0;
                               VAR_RNS_SEQ.Device.PTB290.MaxDev := 0;

                               VAR_RNS_SEQ.Mem.ContainersStop := TRUE;                                                 (* STEP: 47 *)
                               VAR_RNS_SEQ.Mem.ControlInsercion := FALSE;                                              (* STEP: 47 *)
                               VAR_RNS_SEQ.Mem.ControlContinous := FALSE;                                              (* STEP: 47 *)
                               VAR_RNS_SEQ.Mem.PBAbortEnable := FALSE;                                                 (* STEP: 47 PB Abort Sequence Enable*)
                               VAR_RNS_SEQ.Mem.PBStopEnable := TRUE;                                                   (* STEP: 47 PB Stop Sequence Enable*)
                               VAR_RNS_SEQ.Mem.PBStartEnable := FALSE;                                                 (* STEP: 47 PB Start Sequence Enable*)
                               VAR_RNS_SEQ.Mem.ByPassed := FALSE;                                                      (* STEP: 47 *)
                               VAR_RNS_SEQ.Mem.InsercionDevice := FALSE;                                               (* STEP: 47 *)
                               VAR_RNS_SEQ.Mem.AirTreatmentControl := FALSE;                                           (* STEP: 47 *)
                               VAR_RNS_SEQ.Mem.WaterTreatmentControl := FALSE;                                         (* STEP: 47 *)
                               VAR_RNS_SEQ.Mem.SpeedReductionControl := FALSE;                                         (* STEP: 47 *)
                               VAR_RNS_SEQ.Mem.ByPassRequest := FALSE;                                                 (* STEP: 47 *)
                               VAR_RNS_SEQ.Mem.CopAfterCipRequest := FALSE;                                            (* STEP: 47 *)
                               VAR_RNS_SEQ.Mem.NoBoNoSprayInsercion := FALSE;                                          (* STEP: 47 *)

                               VAR_RNS_SEQ.ITC.WTT_ProductRequest := TRUE;                                             (* STEP: 47 *)
                               VAR_RNS_SEQ.ITC.WTT_ProductionRunning := FALSE;                                         (* STEP: 47 *)

                       48: (* CIP - Cycle End *)

                               VAR_RNS_SEQ.Device.AVB224.AutoCnd := TRUE;                                              (* STEP: 48 AVB224*)
                               VAR_RNS_SEQ.Device.AVB224.EnableCnd := FALSE;
                               VAR_RNS_SEQ.Device.AVB228.AutoCnd := FALSE;                                             (* STEP: 48 AVB228*)
                               VAR_RNS_SEQ.Device.AVB228.EnableCnd := FALSE;
                               VAR_RNS_SEQ.Device.AVB234.AutoCnd := FALSE;                                             (* STEP: 48 AVB234*)
                               VAR_RNS_SEQ.Device.AVB234.EnableCnd := FALSE;
                               VAR_RNS_SEQ.Device.AVB261.AutoCnd := FALSE;                                             (* STEP: 48 AVB261*)
                               VAR_RNS_SEQ.Device.AVB261.EnableCnd := FALSE;
                               VAR_RNS_SEQ.Device.AVB264.AutoCnd := FALSE;                                             (* STEP: 48 AVB264*)
                               VAR_RNS_SEQ.Device.AVB264.EnableCnd := FALSE;
                               VAR_RNS_SEQ.Device.AVB265.AutoCnd := FALSE;                                             (* STEP: 48 AVB265*)
                               VAR_RNS_SEQ.Device.AVB265.EnableCnd := FALSE;
                               VAR_RNS_SEQ.Device.AVB266.AutoCnd := TRUE;                                              (* STEP: 48 AVB266*)
                               VAR_RNS_SEQ.Device.AVB266.EnableCnd := FALSE;
                               VAR_RNS_SEQ.Device.AVB267.AutoCnd := TRUE;                                              (* STEP: 48 AVB267*)
                               VAR_RNS_SEQ.Device.AVB267.EnableCnd := FALSE;
                               VAR_RNS_SEQ.Device.AVB268.AutoCnd := TRUE;                                              (* STEP: 48 AVB268*)
                               VAR_RNS_SEQ.Device.AVB268.EnableCnd := FALSE;
                               VAR_RNS_SEQ.Device.AVB273.AutoCnd := FALSE;                                             (* STEP: 48 AVB273*)
                               VAR_RNS_SEQ.Device.AVB273.EnableCnd := FALSE;
                               VAR_RNS_SEQ.Device.AVB294.AutoCnd := FALSE;                                             (* STEP: 48 AVB294*)
                               VAR_RNS_SEQ.Device.AVB294.EnableCnd := FALSE;

                               VAR_RNS_SEQ.Device.PPB209_PID.PID_Enable := FALSE;                                      (* STEP: 48 PPB209*)
                               VAR_RNS_SEQ.Device.PPB209_PID.PID_Mode := FALSE;
                               VAR_RNS_SEQ.Device.PPB209_PID.Auto_SP_Value := 0;
                               VAR_RNS_SEQ.Device.PPB209_PID.FIX_Value := 0;

                               VAR_RNS_SEQ.Device.RVB202_PID.PID_Enable := TRUE;                                       (* STEP: 48 *)
                               VAR_RNS_SEQ.Device.RVB202_PID.PID_Mode := FALSE;
                               VAR_RNS_SEQ.Device.RVB202_PID.Auto_SP_Value := 0;
                               VAR_RNS_SEQ.Device.RVB202_PID.FIX_Value := HMI_PAM_1._093;

                               VAR_RNS_SEQ.Device.FSB220.ALR := FALSE;                                                 (* STEP: 48 FSB220*)
                               VAR_RNS_SEQ.Device.FSB220.WAIT_OFF := FALSE;
                               VAR_RNS_SEQ.Device.FSB220.WAIT_ON := FALSE;

                               VAR_RNS_SEQ.Device.LSB209.ALR := FALSE;                                                 (* STEP: 48 LSB209*)
                               VAR_RNS_SEQ.Device.LSB209.WAIT_OFF := FALSE;
                               VAR_RNS_SEQ.Device.LSB209.WAIT_ON := FALSE;

                               VAR_RNS_SEQ.Device.LSB210.ALR := FALSE;                                                 (* STEP: 48 LSB210*)
                               VAR_RNS_SEQ.Device.LSB210.WAIT_OFF := FALSE;
                               VAR_RNS_SEQ.Device.LSB210.WAIT_ON := FALSE;

                               VAR_RNS_SEQ.Device.LSB299.ALR := FALSE;                                                 (* STEP: 48 *)
                               VAR_RNS_SEQ.Device.LSB299.WAIT_OFF := FALSE;
                               VAR_RNS_SEQ.Device.LSB299.WAIT_ON := FALSE;

                               VAR_RNS_SEQ.Device.FSB201.ALR := FALSE;                                                 (* STEP: 48 FSB201*)
                               VAR_RNS_SEQ.Device.FSB201.WAIT_OFF := FALSE;
                               VAR_RNS_SEQ.Device.FSB201.WAIT_ON := FALSE;

                               VAR_RNS_SEQ.Device.FTB201.ALR_HighLimitEn := FALSE;                                     (* STEP: 48 FTB201*)
                               VAR_RNS_SEQ.Device.FTB201.ALR_HighLimitSP := 0;
                               VAR_RNS_SEQ.Device.FTB201.ALR_LowLimitEn := FALSE;
                               VAR_RNS_SEQ.Device.FTB201.ALR_LowLimitSP := 0;
                               VAR_RNS_SEQ.Device.FTB201.SP := 0;
                               VAR_RNS_SEQ.Device.FTB201.CMP := 0;
                               VAR_RNS_SEQ.Device.FTB201.MinDev := 0;
                               VAR_RNS_SEQ.Device.FTB201.MaxDev := 0;

                               VAR_RNS_SEQ.Device.FTB202.ALR_HighLimitEn := FALSE;                                     (* STEP: 48 FTB202*)
                               VAR_RNS_SEQ.Device.FTB202.ALR_HighLimitSP := 0;
                               VAR_RNS_SEQ.Device.FTB202.ALR_LowLimitEn := FALSE;
                               VAR_RNS_SEQ.Device.FTB202.ALR_LowLimitSP := 0;
                               VAR_RNS_SEQ.Device.FTB202.SP := 0;
                               VAR_RNS_SEQ.Device.FTB202.CMP := 0;
                               VAR_RNS_SEQ.Device.FTB202.MinDev := 0;
                               VAR_RNS_SEQ.Device.FTB202.MaxDev := 0;

                               VAR_RNS_SEQ.Device.PTB220.ALR_HighLimitEn := FALSE;                                     (* STEP: 48 PTB220*)
                               VAR_RNS_SEQ.Device.PTB220.ALR_HighLimitSP := 0;
                               VAR_RNS_SEQ.Device.PTB220.ALR_LowLimitEn := FALSE;
                               VAR_RNS_SEQ.Device.PTB220.ALR_LowLimitSP := 0;
                               VAR_RNS_SEQ.Device.PTB220.SP := 0;
                               VAR_RNS_SEQ.Device.PTB220.CMP := 0;
                               VAR_RNS_SEQ.Device.PTB220.MinDev := 0;
                               VAR_RNS_SEQ.Device.PTB220.MaxDev := 0;

                               VAR_RNS_SEQ.Device.PTB270.ALR_HighLimitEn := FALSE;                                     (* STEP: 48 PTB270*)
                               VAR_RNS_SEQ.Device.PTB270.ALR_HighLimitSP := 0;
                               VAR_RNS_SEQ.Device.PTB270.ALR_LowLimitEn := FALSE;
                               VAR_RNS_SEQ.Device.PTB270.ALR_LowLimitSP := 0;
                               VAR_RNS_SEQ.Device.PTB270.SP := 0;
                               VAR_RNS_SEQ.Device.PTB270.CMP := 0;
                               VAR_RNS_SEQ.Device.PTB270.MinDev := 0;
                               VAR_RNS_SEQ.Device.PTB270.MaxDev := 0;

                               VAR_RNS_SEQ.Device.LTB202.ALR_HighLimitEn := FALSE;                                     (* STEP: 48 LTB202*)
                               VAR_RNS_SEQ.Device.LTB202.ALR_HighLimitSP := 0;
                               VAR_RNS_SEQ.Device.LTB202.ALR_LowLimitEn := FALSE;
                               VAR_RNS_SEQ.Device.LTB202.ALR_LowLimitSP := 0;
                               VAR_RNS_SEQ.Device.LTB202.SP := 0;
                               VAR_RNS_SEQ.Device.LTB202.CMP := 0;
                               VAR_RNS_SEQ.Device.LTB202.MinDev := 0;
                               VAR_RNS_SEQ.Device.LTB202.MaxDev := 0;

                               VAR_RNS_SEQ.Device.PTB290.ALR_HighLimitEn := FALSE;                                     (* STEP: 48 PTB290*)
                               VAR_RNS_SEQ.Device.PTB290.ALR_HighLimitSP := 0;
                               VAR_RNS_SEQ.Device.PTB290.ALR_LowLimitEn := FALSE;
                               VAR_RNS_SEQ.Device.PTB290.ALR_LowLimitSP := 0;
                               VAR_RNS_SEQ.Device.PTB290.SP := 0;
                               VAR_RNS_SEQ.Device.PTB290.CMP := 0;
                               VAR_RNS_SEQ.Device.PTB290.MinDev := 0;
                               VAR_RNS_SEQ.Device.PTB290.MaxDev := 0;

                               VAR_RNS_SEQ.Mem.ContainersStop := FALSE;                                                (* STEP: 48 *)
                               VAR_RNS_SEQ.Mem.ControlInsercion := FALSE;                                              (* STEP: 48 *)
                               VAR_RNS_SEQ.Mem.ControlContinous := FALSE;                                              (* STEP: 48 *)
                               VAR_RNS_SEQ.Mem.PBAbortEnable := FALSE;                                                 (* STEP: 48 PB Abort Sequence Enable*)
                               VAR_RNS_SEQ.Mem.PBStopEnable := FALSE;                                                  (* STEP: 48 PB Stop Sequence Enable*)
                               VAR_RNS_SEQ.Mem.PBStartEnable := FALSE;                                                 (* STEP: 48 PB Start Sequence Enable*)
                               VAR_RNS_SEQ.Mem.ByPassed := FALSE;                                                      (* STEP: 48 *)
                               VAR_RNS_SEQ.Mem.InsercionDevice := FALSE;                                               (* STEP: 48 *)
                               VAR_RNS_SEQ.Mem.AirTreatmentControl := FALSE;                                           (* STEP: 48 *)
                               VAR_RNS_SEQ.Mem.WaterTreatmentControl := FALSE;                                         (* STEP: 48 *)
                               VAR_RNS_SEQ.Mem.SpeedReductionControl := FALSE;                                         (* STEP: 48 *)
                               VAR_RNS_SEQ.Mem.ByPassRequest := FALSE;                                                 (* STEP: 48 *)
                               VAR_RNS_SEQ.Mem.CopAfterCipRequest := FALSE;                                            (* STEP: 48 *)
                               VAR_RNS_SEQ.Mem.NoBoNoSprayInsercion := FALSE;                                          (* STEP: 48 *)

                               VAR_RNS_SEQ.ITC.WTT_ProductRequest := TRUE;                                             (* STEP: 48 *)
                               VAR_RNS_SEQ.ITC.WTT_ProductionRunning := FALSE;                                         (* STEP: 48 *)

                       49: (* CIP - Stopped *)

                               VAR_RNS_SEQ.Device.AVB224.AutoCnd := TRUE;                                              (* STEP: 49 AVB224*)
                               VAR_RNS_SEQ.Device.AVB224.EnableCnd := FALSE;
                               VAR_RNS_SEQ.Device.AVB228.AutoCnd := TRUE;                                              (* STEP: 49 AVB228*)
                               VAR_RNS_SEQ.Device.AVB228.EnableCnd := FALSE;
                               VAR_RNS_SEQ.Device.AVB234.AutoCnd := FALSE;                                             (* STEP: 49 AVB234*)
                               VAR_RNS_SEQ.Device.AVB234.EnableCnd := FALSE;
                               VAR_RNS_SEQ.Device.AVB261.AutoCnd := FALSE;                                             (* STEP: 49 AVB261*)
                               VAR_RNS_SEQ.Device.AVB261.EnableCnd := FALSE;
                               VAR_RNS_SEQ.Device.AVB264.AutoCnd := FALSE;                                             (* STEP: 49 AVB264*)
                               VAR_RNS_SEQ.Device.AVB264.EnableCnd := FALSE;
                               VAR_RNS_SEQ.Device.AVB265.AutoCnd := FALSE;                                             (* STEP: 49 AVB265*)
                               VAR_RNS_SEQ.Device.AVB265.EnableCnd := FALSE;
                               VAR_RNS_SEQ.Device.AVB266.AutoCnd := TRUE;                                              (* STEP: 49 AVB266*)
                               VAR_RNS_SEQ.Device.AVB266.EnableCnd := FALSE;
                               VAR_RNS_SEQ.Device.AVB267.AutoCnd := FALSE;                                             (* STEP: 49 AVB267*)
                               VAR_RNS_SEQ.Device.AVB267.EnableCnd := FALSE;
                               VAR_RNS_SEQ.Device.AVB268.AutoCnd := FALSE;                                             (* STEP: 49 AVB268*)
                               VAR_RNS_SEQ.Device.AVB268.EnableCnd := FALSE;
                               VAR_RNS_SEQ.Device.AVB273.AutoCnd := FALSE;                                             (* STEP: 49 AVB273*)
                               VAR_RNS_SEQ.Device.AVB273.EnableCnd := FALSE;
                               VAR_RNS_SEQ.Device.AVB294.AutoCnd := FALSE;                                             (* STEP: 49 AVB294*)
                               VAR_RNS_SEQ.Device.AVB294.EnableCnd := FALSE;

                               VAR_RNS_SEQ.Device.PPB209_PID.PID_Enable := FALSE;                                      (* STEP: 49 PPB209*)
                               VAR_RNS_SEQ.Device.PPB209_PID.PID_Mode := FALSE;
                               VAR_RNS_SEQ.Device.PPB209_PID.Auto_SP_Value := 0;
                               VAR_RNS_SEQ.Device.PPB209_PID.FIX_Value := 0;

                               VAR_RNS_SEQ.Device.RVB202_PID.PID_Enable := FALSE;                                      (* STEP: 49 *)
                               VAR_RNS_SEQ.Device.RVB202_PID.PID_Mode := FALSE;
                               VAR_RNS_SEQ.Device.RVB202_PID.Auto_SP_Value := 0;
                               VAR_RNS_SEQ.Device.RVB202_PID.FIX_Value := 0;

                               VAR_RNS_SEQ.Device.FSB220.ALR := FALSE;                                                 (* STEP: 49 FSB220*)
                               VAR_RNS_SEQ.Device.FSB220.WAIT_OFF := FALSE;
                               VAR_RNS_SEQ.Device.FSB220.WAIT_ON := FALSE;

                               VAR_RNS_SEQ.Device.LSB209.ALR := FALSE;                                                 (* STEP: 49 LSB209*)
                               VAR_RNS_SEQ.Device.LSB209.WAIT_OFF := FALSE;
                               VAR_RNS_SEQ.Device.LSB209.WAIT_ON := FALSE;

                               VAR_RNS_SEQ.Device.LSB210.ALR := FALSE;                                                 (* STEP: 49 LSB210*)
                               VAR_RNS_SEQ.Device.LSB210.WAIT_OFF := FALSE;
                               VAR_RNS_SEQ.Device.LSB210.WAIT_ON := FALSE;

                               VAR_RNS_SEQ.Device.LSB299.ALR := FALSE;                                                 (* STEP: 49 *)
                               VAR_RNS_SEQ.Device.LSB299.WAIT_OFF := FALSE;
                               VAR_RNS_SEQ.Device.LSB299.WAIT_ON := FALSE;

                               VAR_RNS_SEQ.Device.FSB201.ALR := FALSE;                                                 (* STEP: 49 FSB201*)
                               VAR_RNS_SEQ.Device.FSB201.WAIT_OFF := FALSE;
                               VAR_RNS_SEQ.Device.FSB201.WAIT_ON := FALSE;

                               VAR_RNS_SEQ.Device.FTB201.ALR_HighLimitEn := FALSE;                                     (* STEP: 49 FTB201*)
                               VAR_RNS_SEQ.Device.FTB201.ALR_HighLimitSP := 0;
                               VAR_RNS_SEQ.Device.FTB201.ALR_LowLimitEn := FALSE;
                               VAR_RNS_SEQ.Device.FTB201.ALR_LowLimitSP := 0;
                               VAR_RNS_SEQ.Device.FTB201.SP := 0;
                               VAR_RNS_SEQ.Device.FTB201.CMP := 0;
                               VAR_RNS_SEQ.Device.FTB201.MinDev := 0;
                               VAR_RNS_SEQ.Device.FTB201.MaxDev := 0;

                               VAR_RNS_SEQ.Device.FTB202.ALR_HighLimitEn := FALSE;                                     (* STEP: 49 FTB202*)
                               VAR_RNS_SEQ.Device.FTB202.ALR_HighLimitSP := 0;
                               VAR_RNS_SEQ.Device.FTB202.ALR_LowLimitEn := FALSE;
                               VAR_RNS_SEQ.Device.FTB202.ALR_LowLimitSP := 0;
                               VAR_RNS_SEQ.Device.FTB202.SP := 0;
                               VAR_RNS_SEQ.Device.FTB202.CMP := 0;
                               VAR_RNS_SEQ.Device.FTB202.MinDev := 0;
                               VAR_RNS_SEQ.Device.FTB202.MaxDev := 0;

                               VAR_RNS_SEQ.Device.PTB220.ALR_HighLimitEn := FALSE;                                     (* STEP: 49 PTB220*)
                               VAR_RNS_SEQ.Device.PTB220.ALR_HighLimitSP := 0;
                               VAR_RNS_SEQ.Device.PTB220.ALR_LowLimitEn := FALSE;
                               VAR_RNS_SEQ.Device.PTB220.ALR_LowLimitSP := 0;
                               VAR_RNS_SEQ.Device.PTB220.SP := 0;
                               VAR_RNS_SEQ.Device.PTB220.CMP := 0;
                               VAR_RNS_SEQ.Device.PTB220.MinDev := 0;
                               VAR_RNS_SEQ.Device.PTB220.MaxDev := 0;

                               VAR_RNS_SEQ.Device.PTB270.ALR_HighLimitEn := FALSE;                                     (* STEP: 49 PTB270*)
                               VAR_RNS_SEQ.Device.PTB270.ALR_HighLimitSP := 0;
                               VAR_RNS_SEQ.Device.PTB270.ALR_LowLimitEn := FALSE;
                               VAR_RNS_SEQ.Device.PTB270.ALR_LowLimitSP := 0;
                               VAR_RNS_SEQ.Device.PTB270.SP := 0;
                               VAR_RNS_SEQ.Device.PTB270.CMP := 0;
                               VAR_RNS_SEQ.Device.PTB270.MinDev := 0;
                               VAR_RNS_SEQ.Device.PTB270.MaxDev := 0;

                               VAR_RNS_SEQ.Device.LTB202.ALR_HighLimitEn := FALSE;                                     (* STEP: 49 LTB202*)
                               VAR_RNS_SEQ.Device.LTB202.ALR_HighLimitSP := 0;
                               VAR_RNS_SEQ.Device.LTB202.ALR_LowLimitEn := FALSE;
                               VAR_RNS_SEQ.Device.LTB202.ALR_LowLimitSP := 0;
                               VAR_RNS_SEQ.Device.LTB202.SP := 0;
                               VAR_RNS_SEQ.Device.LTB202.CMP := 0;
                               VAR_RNS_SEQ.Device.LTB202.MinDev := 0;
                               VAR_RNS_SEQ.Device.LTB202.MaxDev := 0;

                               VAR_RNS_SEQ.Device.PTB290.ALR_HighLimitEn := FALSE;                                     (* STEP: 49 PTB290*)
                               VAR_RNS_SEQ.Device.PTB290.ALR_HighLimitSP := 0;
                               VAR_RNS_SEQ.Device.PTB290.ALR_LowLimitEn := FALSE;
                               VAR_RNS_SEQ.Device.PTB290.ALR_LowLimitSP := 0;
                               VAR_RNS_SEQ.Device.PTB290.SP := 0;
                               VAR_RNS_SEQ.Device.PTB290.CMP := 0;
                               VAR_RNS_SEQ.Device.PTB290.MinDev := 0;
                               VAR_RNS_SEQ.Device.PTB290.MaxDev := 0;

                               VAR_RNS_SEQ.Mem.ContainersStop := TRUE;                                                 (* STEP: 49 *)
                               VAR_RNS_SEQ.Mem.ControlInsercion := FALSE;                                              (* STEP: 49 *)
                               VAR_RNS_SEQ.Mem.ControlContinous := FALSE;                                              (* STEP: 49 *)
                               VAR_RNS_SEQ.Mem.PBAbortEnable := FALSE;                                                 (* STEP: 49 PB Abort Sequence Enable*)
                               VAR_RNS_SEQ.Mem.PBStopEnable := TRUE;                                                   (* STEP: 49 PB Stop Sequence Enable*)
                               VAR_RNS_SEQ.Mem.PBStartEnable := FALSE;                                                 (* STEP: 49 PB Start Sequence Enable*)
                               VAR_RNS_SEQ.Mem.ByPassed := FALSE;                                                      (* STEP: 49 *)
                               VAR_RNS_SEQ.Mem.InsercionDevice := FALSE;                                               (* STEP: 49 *)
                               VAR_RNS_SEQ.Mem.AirTreatmentControl := FALSE;                                           (* STEP: 49 *)
                               VAR_RNS_SEQ.Mem.WaterTreatmentControl := FALSE;                                         (* STEP: 49 *)
                               VAR_RNS_SEQ.Mem.SpeedReductionControl := FALSE;                                          (* STEP: 49 *)
                               VAR_RNS_SEQ.Mem.ByPassRequest := FALSE;                                                 (* STEP: 49 *)
                               VAR_RNS_SEQ.Mem.CopAfterCipRequest := FALSE;                                            (* STEP: 49 *)
                               VAR_RNS_SEQ.Mem.NoBoNoSprayInsercion := FALSE;                                          (* STEP: 49 *)

                               VAR_RNS_SEQ.ITC.WTT_ProductRequest := FALSE;                                            (* STEP: 49 *)
                               VAR_RNS_SEQ.ITC.WTT_ProductionRunning := FALSE;                                         (* STEP: 49 *)

                       50: (* DRAINING - Tank and circuit emptying *)

                               VAR_RNS_SEQ.Device.AVB224.AutoCnd := TRUE;                                              (* STEP: 50 AVB224*)
                               VAR_RNS_SEQ.Device.AVB224.EnableCnd := FALSE;
                               VAR_RNS_SEQ.Device.AVB228.AutoCnd := FALSE;                                             (* STEP: 50 AVB228*)
                               VAR_RNS_SEQ.Device.AVB228.EnableCnd := FALSE;
                               VAR_RNS_SEQ.Device.AVB234.AutoCnd := TRUE;                                              (* STEP: 50 AVB234*)
                               VAR_RNS_SEQ.Device.AVB234.EnableCnd := FALSE;
                               VAR_RNS_SEQ.Device.AVB261.AutoCnd := FALSE;                                             (* STEP: 50 AVB261*)
                               VAR_RNS_SEQ.Device.AVB261.EnableCnd := FALSE;
                               VAR_RNS_SEQ.Device.AVB264.AutoCnd := FALSE;                                             (* STEP: 50 AVB264*)
                               VAR_RNS_SEQ.Device.AVB264.EnableCnd := FALSE;
                               VAR_RNS_SEQ.Device.AVB265.AutoCnd := FALSE;                                             (* STEP: 50 AVB265*)
                               VAR_RNS_SEQ.Device.AVB265.EnableCnd := FALSE;
                               VAR_RNS_SEQ.Device.AVB266.AutoCnd := TRUE;                                              (* STEP: 50 AVB266*)
                               VAR_RNS_SEQ.Device.AVB266.EnableCnd := FALSE;
                               VAR_RNS_SEQ.Device.AVB267.AutoCnd := TRUE;                                              (* STEP: 50 AVB267*)
                               VAR_RNS_SEQ.Device.AVB267.EnableCnd := FALSE;
                               VAR_RNS_SEQ.Device.AVB268.AutoCnd := TRUE;                                              (* STEP: 50 AVB268*)
                               VAR_RNS_SEQ.Device.AVB268.EnableCnd := FALSE;
                               VAR_RNS_SEQ.Device.AVB273.AutoCnd := FALSE;                                             (* STEP: 50 AVB273*)
                               VAR_RNS_SEQ.Device.AVB273.EnableCnd := FALSE;
                               VAR_RNS_SEQ.Device.AVB294.AutoCnd := FALSE;                                             (* STEP: 50 AVB294*)
                               VAR_RNS_SEQ.Device.AVB294.EnableCnd := FALSE;

                               VAR_RNS_SEQ.Device.PPB209_PID.PID_Enable := FALSE;                                      (* STEP: 50 PPB209*)
                               VAR_RNS_SEQ.Device.PPB209_PID.PID_Mode := FALSE;
                               VAR_RNS_SEQ.Device.PPB209_PID.Auto_SP_Value := 0;
                               VAR_RNS_SEQ.Device.PPB209_PID.FIX_Value := 0;

                               VAR_RNS_SEQ.Device.RVB202_PID.PID_Enable := FALSE;                                      (* STEP: 50 *)
                               VAR_RNS_SEQ.Device.RVB202_PID.PID_Mode := FALSE;
                               VAR_RNS_SEQ.Device.RVB202_PID.Auto_SP_Value := 0;
                               VAR_RNS_SEQ.Device.RVB202_PID.FIX_Value := 0;

                               VAR_RNS_SEQ.Device.FSB220.ALR := FALSE;                                                 (* STEP: 50 FSB220*)
                               VAR_RNS_SEQ.Device.FSB220.WAIT_OFF := FALSE;
                               VAR_RNS_SEQ.Device.FSB220.WAIT_ON := FALSE;

                               VAR_RNS_SEQ.Device.LSB209.ALR := FALSE;                                                 (* STEP: 50 LSB209*)
                               VAR_RNS_SEQ.Device.LSB209.WAIT_OFF := FALSE;
                               VAR_RNS_SEQ.Device.LSB209.WAIT_ON := FALSE;

                               VAR_RNS_SEQ.Device.LSB210.ALR := FALSE;                                                 (* STEP: 50 LSB210*)
                               VAR_RNS_SEQ.Device.LSB210.WAIT_OFF := FALSE;
                               VAR_RNS_SEQ.Device.LSB210.WAIT_ON := FALSE;

                               VAR_RNS_SEQ.Device.LSB299.ALR := FALSE;                                                 (* STEP: 50 *)
                               VAR_RNS_SEQ.Device.LSB299.WAIT_OFF := FALSE;
                               VAR_RNS_SEQ.Device.LSB299.WAIT_ON := FALSE;

                               VAR_RNS_SEQ.Device.FSB201.ALR := FALSE;                                                 (* STEP: 50 FSB201*)
                               VAR_RNS_SEQ.Device.FSB201.WAIT_OFF := FALSE;
                               VAR_RNS_SEQ.Device.FSB201.WAIT_ON := FALSE;

                               VAR_RNS_SEQ.Device.FTB201.ALR_HighLimitEn := FALSE;                                     (* STEP: 50 FTB201*)
                               VAR_RNS_SEQ.Device.FTB201.ALR_HighLimitSP := 0;
                               VAR_RNS_SEQ.Device.FTB201.ALR_LowLimitEn := FALSE;
                               VAR_RNS_SEQ.Device.FTB201.ALR_LowLimitSP := 0;
                               VAR_RNS_SEQ.Device.FTB201.SP := 0;
                               VAR_RNS_SEQ.Device.FTB201.CMP := 0;
                               VAR_RNS_SEQ.Device.FTB201.MinDev := 0;
                               VAR_RNS_SEQ.Device.FTB201.MaxDev := 0;

                               VAR_RNS_SEQ.Device.FTB202.ALR_HighLimitEn := FALSE;                                     (* STEP: 50 FTB202*)
                               VAR_RNS_SEQ.Device.FTB202.ALR_HighLimitSP := 0;
                               VAR_RNS_SEQ.Device.FTB202.ALR_LowLimitEn := FALSE;
                               VAR_RNS_SEQ.Device.FTB202.ALR_LowLimitSP := 0;
                               VAR_RNS_SEQ.Device.FTB202.SP := 0;
                               VAR_RNS_SEQ.Device.FTB202.CMP := 0;
                               VAR_RNS_SEQ.Device.FTB202.MinDev := 0;
                               VAR_RNS_SEQ.Device.FTB202.MaxDev := 0;

                               VAR_RNS_SEQ.Device.PTB220.ALR_HighLimitEn := FALSE;                                     (* STEP: 50 PTB220*)
                               VAR_RNS_SEQ.Device.PTB220.ALR_HighLimitSP := 0;
                               VAR_RNS_SEQ.Device.PTB220.ALR_LowLimitEn := FALSE;
                               VAR_RNS_SEQ.Device.PTB220.ALR_LowLimitSP := 0;
                               VAR_RNS_SEQ.Device.PTB220.SP := 0;
                               VAR_RNS_SEQ.Device.PTB220.CMP := 0;
                               VAR_RNS_SEQ.Device.PTB220.MinDev := 0;
                               VAR_RNS_SEQ.Device.PTB220.MaxDev := 0;

                               VAR_RNS_SEQ.Device.PTB270.ALR_HighLimitEn := FALSE;                                     (* STEP: 50 PTB270*)
                               VAR_RNS_SEQ.Device.PTB270.ALR_HighLimitSP := 0;
                               VAR_RNS_SEQ.Device.PTB270.ALR_LowLimitEn := FALSE;
                               VAR_RNS_SEQ.Device.PTB270.ALR_LowLimitSP := 0;
                               VAR_RNS_SEQ.Device.PTB270.SP := 0;
                               VAR_RNS_SEQ.Device.PTB270.CMP := 0;
                               VAR_RNS_SEQ.Device.PTB270.MinDev := 0;
                               VAR_RNS_SEQ.Device.PTB270.MaxDev := 0;

                               VAR_RNS_SEQ.Device.LTB202.ALR_HighLimitEn := FALSE;                                     (* STEP: 50 LTB202*)
                               VAR_RNS_SEQ.Device.LTB202.ALR_HighLimitSP := 0;
                               VAR_RNS_SEQ.Device.LTB202.ALR_LowLimitEn := FALSE;
                               VAR_RNS_SEQ.Device.LTB202.ALR_LowLimitSP := 0;
                               VAR_RNS_SEQ.Device.LTB202.SP := 0;
                               VAR_RNS_SEQ.Device.LTB202.CMP := 0;
                               VAR_RNS_SEQ.Device.LTB202.MinDev := 0;
                               VAR_RNS_SEQ.Device.LTB202.MaxDev := 0;

                               VAR_RNS_SEQ.Device.PTB290.ALR_HighLimitEn := FALSE;                                     (* STEP: 50 PTB290*)
                               VAR_RNS_SEQ.Device.PTB290.ALR_HighLimitSP := 0;
                               VAR_RNS_SEQ.Device.PTB290.ALR_LowLimitEn := FALSE;
                               VAR_RNS_SEQ.Device.PTB290.ALR_LowLimitSP := 0;
                               VAR_RNS_SEQ.Device.PTB290.SP := 0;
                               VAR_RNS_SEQ.Device.PTB290.CMP := 0;
                               VAR_RNS_SEQ.Device.PTB290.MinDev := 0;
                               VAR_RNS_SEQ.Device.PTB290.MaxDev := 0;

                               VAR_RNS_SEQ.Mem.ContainersStop := TRUE;                                                 (* STEP: 50 *)
                               VAR_RNS_SEQ.Mem.ControlInsercion := FALSE;                                              (* STEP: 50 *)
                               VAR_RNS_SEQ.Mem.ControlContinous := FALSE;                                              (* STEP: 50 *)
                               VAR_RNS_SEQ.Mem.PBAbortEnable := FALSE;                                                 (* STEP: 50 PB Abort Sequence Enable*)
                               VAR_RNS_SEQ.Mem.PBStopEnable := TRUE;                                                   (* STEP: 50 PB Stop Sequence Enable*)
                               VAR_RNS_SEQ.Mem.PBStartEnable := FALSE;                                                 (* STEP: 50 PB Start Sequence Enable*)
                               VAR_RNS_SEQ.Mem.ByPassed := FALSE;                                                      (* STEP: 50 *)
                               VAR_RNS_SEQ.Mem.InsercionDevice := FALSE;                                               (* STEP: 50 *)
                               VAR_RNS_SEQ.Mem.AirTreatmentControl := FALSE;                                           (* STEP: 50 *)
                               VAR_RNS_SEQ.Mem.WaterTreatmentControl := FALSE;                                         (* STEP: 50 *)
                               VAR_RNS_SEQ.Mem.SpeedReductionControl := FALSE;                                         (* STEP: 50 *)
                               VAR_RNS_SEQ.Mem.ByPassRequest := FALSE;                                                 (* STEP: 50 *)
                               VAR_RNS_SEQ.Mem.CopAfterCipRequest := FALSE;                                            (* STEP: 50 *)
                               VAR_RNS_SEQ.Mem.NoBoNoSprayInsercion := FALSE;                                          (* STEP: 50 *)

                               VAR_RNS_SEQ.ITC.WTT_ProductRequest := FALSE;                                            (* STEP: 50 *)
                               VAR_RNS_SEQ.ITC.WTT_ProductionRunning := FALSE;                                         (* STEP: 50 *)

                       51: (* DRAINING - End drain cycle *)

                               VAR_RNS_SEQ.Device.AVB224.AutoCnd := TRUE;                                              (* STEP: 51 AVB224*)
                               VAR_RNS_SEQ.Device.AVB224.EnableCnd := FALSE;
                               VAR_RNS_SEQ.Device.AVB228.AutoCnd := FALSE;                                             (* STEP: 51 AVB228*)
                               VAR_RNS_SEQ.Device.AVB228.EnableCnd := FALSE;
                               VAR_RNS_SEQ.Device.AVB234.AutoCnd := TRUE;                                              (* STEP: 51 AVB234*)
                               VAR_RNS_SEQ.Device.AVB234.EnableCnd := FALSE;
                               VAR_RNS_SEQ.Device.AVB261.AutoCnd := FALSE;                                             (* STEP: 51 AVB261*)
                               VAR_RNS_SEQ.Device.AVB261.EnableCnd := FALSE;
                               VAR_RNS_SEQ.Device.AVB264.AutoCnd := FALSE;                                             (* STEP: 51 AVB264*)
                               VAR_RNS_SEQ.Device.AVB264.EnableCnd := FALSE;
                               VAR_RNS_SEQ.Device.AVB265.AutoCnd := FALSE;                                             (* STEP: 51 AVB265*)
                               VAR_RNS_SEQ.Device.AVB265.EnableCnd := FALSE;
                               VAR_RNS_SEQ.Device.AVB266.AutoCnd := TRUE;                                              (* STEP: 51 AVB266*)
                               VAR_RNS_SEQ.Device.AVB266.EnableCnd := FALSE;
                               VAR_RNS_SEQ.Device.AVB267.AutoCnd := TRUE;                                              (* STEP: 51 AVB267*)
                               VAR_RNS_SEQ.Device.AVB267.EnableCnd := FALSE;
                               VAR_RNS_SEQ.Device.AVB268.AutoCnd := TRUE;                                              (* STEP: 51 AVB268*)
                               VAR_RNS_SEQ.Device.AVB268.EnableCnd := FALSE;
                               VAR_RNS_SEQ.Device.AVB273.AutoCnd := FALSE;                                             (* STEP: 51 AVB273*)
                               VAR_RNS_SEQ.Device.AVB273.EnableCnd := FALSE;
                               VAR_RNS_SEQ.Device.AVB294.AutoCnd := FALSE;                                             (* STEP: 51 AVB294*)
                               VAR_RNS_SEQ.Device.AVB294.EnableCnd := FALSE;

                               VAR_RNS_SEQ.Device.PPB209_PID.PID_Enable := FALSE;                                      (* STEP: 51 PPB209*)
                               VAR_RNS_SEQ.Device.PPB209_PID.PID_Mode := FALSE;
                               VAR_RNS_SEQ.Device.PPB209_PID.Auto_SP_Value := 0;
                               VAR_RNS_SEQ.Device.PPB209_PID.FIX_Value := 0;

                               VAR_RNS_SEQ.Device.RVB202_PID.PID_Enable := FALSE;                                      (* STEP: 51 *)
                               VAR_RNS_SEQ.Device.RVB202_PID.PID_Mode := FALSE;
                               VAR_RNS_SEQ.Device.RVB202_PID.Auto_SP_Value := 0;
                               VAR_RNS_SEQ.Device.RVB202_PID.FIX_Value := 0;

                               VAR_RNS_SEQ.Device.FSB220.ALR := FALSE;                                                 (* STEP: 51 FSB220*)
                               VAR_RNS_SEQ.Device.FSB220.WAIT_OFF := FALSE;
                               VAR_RNS_SEQ.Device.FSB220.WAIT_ON := FALSE;

                               VAR_RNS_SEQ.Device.LSB209.ALR := FALSE;                                                 (* STEP: 51 LSB209*)
                               VAR_RNS_SEQ.Device.LSB209.WAIT_OFF := FALSE;
                               VAR_RNS_SEQ.Device.LSB209.WAIT_ON := FALSE;

                               VAR_RNS_SEQ.Device.LSB210.ALR := FALSE;                                                 (* STEP: 51 LSB210*)
                               VAR_RNS_SEQ.Device.LSB210.WAIT_OFF := FALSE;
                               VAR_RNS_SEQ.Device.LSB210.WAIT_ON := FALSE;

                               VAR_RNS_SEQ.Device.LSB299.ALR := FALSE;                                                 (* STEP: 51 *)
                               VAR_RNS_SEQ.Device.LSB299.WAIT_OFF := FALSE;
                               VAR_RNS_SEQ.Device.LSB299.WAIT_ON := FALSE;

                               VAR_RNS_SEQ.Device.FSB201.ALR := FALSE;                                                 (* STEP: 51 FSB201*)
                               VAR_RNS_SEQ.Device.FSB201.WAIT_OFF := FALSE;
                               VAR_RNS_SEQ.Device.FSB201.WAIT_ON := FALSE;

                               VAR_RNS_SEQ.Device.FTB201.ALR_HighLimitEn := FALSE;                                     (* STEP: 51 FTB201*)
                               VAR_RNS_SEQ.Device.FTB201.ALR_HighLimitSP := 0;
                               VAR_RNS_SEQ.Device.FTB201.ALR_LowLimitEn := FALSE;
                               VAR_RNS_SEQ.Device.FTB201.ALR_LowLimitSP := 0;
                               VAR_RNS_SEQ.Device.FTB201.SP := 0;
                               VAR_RNS_SEQ.Device.FTB201.CMP := 0;
                               VAR_RNS_SEQ.Device.FTB201.MinDev := 0;
                               VAR_RNS_SEQ.Device.FTB201.MaxDev := 0;

                               VAR_RNS_SEQ.Device.FTB202.ALR_HighLimitEn := FALSE;                                     (* STEP: 51 FTB202*)
                               VAR_RNS_SEQ.Device.FTB202.ALR_HighLimitSP := 0;
                               VAR_RNS_SEQ.Device.FTB202.ALR_LowLimitEn := FALSE;
                               VAR_RNS_SEQ.Device.FTB202.ALR_LowLimitSP := 0;
                               VAR_RNS_SEQ.Device.FTB202.SP := 0;
                               VAR_RNS_SEQ.Device.FTB202.CMP := 0;
                               VAR_RNS_SEQ.Device.FTB202.MinDev := 0;
                               VAR_RNS_SEQ.Device.FTB202.MaxDev := 0;

                               VAR_RNS_SEQ.Device.PTB220.ALR_HighLimitEn := FALSE;                                     (* STEP: 51 PTB220*)
                               VAR_RNS_SEQ.Device.PTB220.ALR_HighLimitSP := 0;
                               VAR_RNS_SEQ.Device.PTB220.ALR_LowLimitEn := FALSE;
                               VAR_RNS_SEQ.Device.PTB220.ALR_LowLimitSP := 0;
                               VAR_RNS_SEQ.Device.PTB220.SP := 0;
                               VAR_RNS_SEQ.Device.PTB220.CMP := 0;
                               VAR_RNS_SEQ.Device.PTB220.MinDev := 0;
                               VAR_RNS_SEQ.Device.PTB220.MaxDev := 0;

                               VAR_RNS_SEQ.Device.PTB270.ALR_HighLimitEn := FALSE;                                     (* STEP: 51 PTB270*)
                               VAR_RNS_SEQ.Device.PTB270.ALR_HighLimitSP := 0;
                               VAR_RNS_SEQ.Device.PTB270.ALR_LowLimitEn := FALSE;
                               VAR_RNS_SEQ.Device.PTB270.ALR_LowLimitSP := 0;
                               VAR_RNS_SEQ.Device.PTB270.SP := 0;
                               VAR_RNS_SEQ.Device.PTB270.CMP := 0;
                               VAR_RNS_SEQ.Device.PTB270.MinDev := 0;
                               VAR_RNS_SEQ.Device.PTB270.MaxDev := 0;

                               VAR_RNS_SEQ.Device.LTB202.ALR_HighLimitEn := FALSE;                                     (* STEP: 51 LTB202*)
                               VAR_RNS_SEQ.Device.LTB202.ALR_HighLimitSP := 0;
                               VAR_RNS_SEQ.Device.LTB202.ALR_LowLimitEn := FALSE;
                               VAR_RNS_SEQ.Device.LTB202.ALR_LowLimitSP := 0;
                               VAR_RNS_SEQ.Device.LTB202.SP := 3;
                               VAR_RNS_SEQ.Device.LTB202.CMP := 1;
                               VAR_RNS_SEQ.Device.LTB202.MinDev := 0;
                               VAR_RNS_SEQ.Device.LTB202.MaxDev := 0;

                               VAR_RNS_SEQ.Device.PTB290.ALR_HighLimitEn := FALSE;                                     (* STEP: 51 PTB290*)
                               VAR_RNS_SEQ.Device.PTB290.ALR_HighLimitSP := 0;
                               VAR_RNS_SEQ.Device.PTB290.ALR_LowLimitEn := FALSE;
                               VAR_RNS_SEQ.Device.PTB290.ALR_LowLimitSP := 0;
                               VAR_RNS_SEQ.Device.PTB290.SP := 0;
                               VAR_RNS_SEQ.Device.PTB290.CMP := 0;
                               VAR_RNS_SEQ.Device.PTB290.MinDev := 0;
                               VAR_RNS_SEQ.Device.PTB290.MaxDev := 0;
```
